Yaskawa INFORM job: A_ROOF_SIDE_0617_2_PAINT_54.JBI

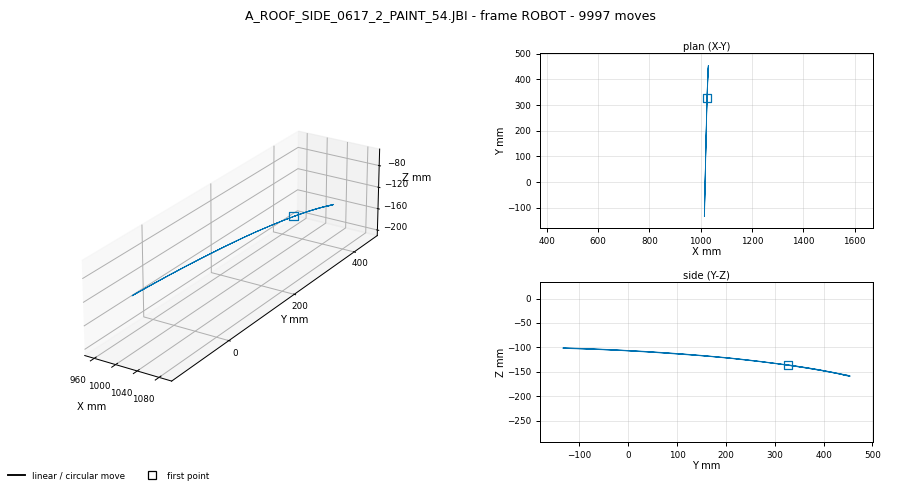
[picture p0: tool path of A_ROOF_SIDE_0617_2_PAINT_54.JBI in frame ROBOT, 9997 of 9997 moves have a stored position in this frame; points joined in program order, loops and branches not executed]
/JOB
//NAME A_ROOF_SIDE_0617_2_PAINT54
//POS
///NPOS 9997,0,0,0,0,0
///TOOL 1
///USER 0
///POSTYPE ROBOT
///RECTAN
///RCONF 1,0,0,0,0,0,0,0,0,0,0,0,0,0,0,0,0,0,0,0,0,0,0,0
C00000=1025.323,327.498,-135.693,171.201,47.894,159.349
C00001=1025.330,327.745,-135.728,171.208,47.893,159.349
C00002=1025.337,327.993,-135.764,171.213,47.892,159.350
C00003=1025.345,328.240,-135.798,171.218,47.891,159.350
C00004=1025.352,328.488,-135.834,171.225,47.891,159.351
C00005=1025.359,328.735,-135.869,171.230,47.890,159.352
C00006=1025.365,328.982,-135.905,171.237,47.889,159.352
C00007=1025.373,329.230,-135.940,171.242,47.888,159.353
C00008=1025.380,329.477,-135.975,171.248,47.888,159.354
C00009=1025.388,329.725,-136.010,171.254,47.886,159.354
C00010=1025.395,329.972,-136.046,171.260,47.886,159.355
C00011=1025.402,330.219,-136.081,171.265,47.885,159.355
C00012=1025.409,330.467,-136.117,171.272,47.885,159.356
C00013=1025.417,330.714,-136.152,171.277,47.884,159.357
C00014=1025.424,330.961,-136.187,171.284,47.883,159.358
C00015=1025.431,331.209,-136.222,171.289,47.883,159.358
C00016=1025.438,331.456,-136.258,171.295,47.882,159.359
C00017=1025.445,331.704,-136.294,171.301,47.881,159.359
C00018=1025.453,331.951,-136.328,171.307,47.880,159.360
C00019=1025.461,332.199,-136.365,171.313,47.880,159.361
C00020=1025.467,332.446,-136.400,171.319,47.880,159.361
C00021=1025.475,332.693,-136.436,171.325,47.878,159.362
C00022=1025.482,332.941,-136.471,171.331,47.878,159.363
C00023=1025.489,333.188,-136.507,171.337,47.877,159.363
C00024=1025.497,333.435,-136.542,171.343,47.877,159.364
C00025=1025.505,333.683,-136.578,171.348,47.876,159.365
C00026=1025.512,333.929,-136.614,171.355,47.876,159.365
C00027=1025.519,334.177,-136.649,171.361,47.875,159.366
C00028=1025.526,334.424,-136.685,171.368,47.875,159.367
C00029=1025.534,334.672,-136.721,171.373,47.874,159.368
C00030=1025.540,334.920,-136.758,171.380,47.873,159.368
C00031=1025.547,335.167,-136.793,171.385,47.873,159.369
C00032=1025.555,335.414,-136.830,171.392,47.873,159.370
C00033=1025.562,335.661,-136.865,171.398,47.872,159.371
C00034=1025.574,336.048,-136.922,171.407,47.871,159.372
C00035=1025.586,336.435,-136.978,171.416,47.871,159.373
C00036=1025.597,336.822,-137.034,171.426,47.870,159.374
C00037=1025.608,337.209,-137.091,171.435,47.869,159.375
C00038=1025.616,337.456,-137.127,171.442,47.869,159.376
C00039=1025.623,337.704,-137.163,171.448,47.869,159.376
C00040=1025.631,337.951,-137.199,171.455,47.868,159.377
C00041=1025.638,338.198,-137.235,171.460,47.868,159.378
C00042=1025.646,338.446,-137.272,171.467,47.867,159.379
C00043=1025.654,338.693,-137.308,171.474,47.867,159.380
C00044=1025.661,338.940,-137.344,171.479,47.866,159.380
C00045=1025.668,339.187,-137.380,171.486,47.866,159.381
C00046=1025.676,339.435,-137.416,171.492,47.866,159.382
C00047=1025.684,339.682,-137.452,171.498,47.865,159.383
C00048=1025.691,339.930,-137.489,171.504,47.865,159.383
C00049=1025.698,340.176,-137.526,171.511,47.865,159.384
C00050=1025.706,340.423,-137.562,171.517,47.865,159.385
C00051=1025.713,340.671,-137.598,171.523,47.864,159.386
C00052=1025.721,340.918,-137.636,171.530,47.864,159.387
C00053=1025.728,341.165,-137.672,171.536,47.864,159.387
C00054=1025.735,341.412,-137.708,171.543,47.864,159.388
C00055=1025.743,341.659,-137.745,171.548,47.863,159.389
C00056=1025.750,341.907,-137.782,171.555,47.863,159.390
C00057=1025.758,342.154,-137.818,171.561,47.863,159.391
C00058=1025.765,342.401,-137.855,171.568,47.863,159.392
C00059=1025.773,342.649,-137.891,171.575,47.862,159.392
C00060=1025.781,342.896,-137.928,171.581,47.863,159.393
C00061=1025.788,343.143,-137.965,171.587,47.862,159.394
C00062=1025.796,343.390,-138.002,171.593,47.862,159.395
C00063=1025.803,343.638,-138.038,171.600,47.862,159.396
C00064=1025.811,343.885,-138.076,171.607,47.861,159.397
C00065=1025.818,344.131,-138.112,171.613,47.862,159.397
C00066=1025.825,344.379,-138.149,171.619,47.861,159.398
C00067=1025.833,344.625,-138.186,171.626,47.861,159.399
C00068=1025.841,344.872,-138.223,171.632,47.861,159.400
C00069=1025.848,345.120,-138.260,171.639,47.861,159.401
C00070=1025.856,345.367,-138.297,171.645,47.861,159.402
C00071=1025.864,345.615,-138.335,171.652,47.861,159.403
C00072=1025.871,345.862,-138.371,171.658,47.860,159.403
C00073=1025.879,346.109,-138.409,171.664,47.861,159.404
C00074=1025.887,346.356,-138.445,171.671,47.861,159.405
C00075=1025.895,346.603,-138.482,171.678,47.860,159.406
C00076=1025.902,346.850,-138.520,171.685,47.860,159.407
C00077=1025.910,347.097,-138.557,171.691,47.861,159.408
C00078=1025.917,347.345,-138.594,171.698,47.860,159.409
C00079=1025.925,347.591,-138.631,171.705,47.860,159.410
C00080=1025.932,347.839,-138.668,171.711,47.861,159.411
C00081=1025.941,348.086,-138.705,171.718,47.861,159.412
C00082=1025.948,348.333,-138.743,171.725,47.860,159.412
C00083=1025.956,348.580,-138.780,171.732,47.860,159.413
C00084=1025.963,348.827,-138.818,171.738,47.861,159.414
C00085=1025.971,349.074,-138.856,171.745,47.861,159.415
C00086=1025.979,349.321,-138.893,171.752,47.861,159.416
C00087=1025.986,349.568,-138.930,171.758,47.861,159.417
C00088=1025.994,349.816,-138.968,171.765,47.861,159.418
C00089=1026.005,350.185,-139.025,171.775,47.861,159.420
C00090=1026.016,350.531,-139.077,171.784,47.861,159.421
C00091=1026.023,350.754,-139.110,171.790,47.862,159.422
C00092=1026.030,350.977,-139.145,171.796,47.862,159.423
C00093=1026.037,351.199,-139.179,171.802,47.862,159.424
C00094=1026.044,351.423,-139.213,171.809,47.862,159.424
C00095=1026.051,351.645,-139.247,171.815,47.862,159.425
C00096=1026.058,351.868,-139.281,171.821,47.863,159.426
C00097=1026.065,352.090,-139.315,171.827,47.863,159.427
C00098=1026.074,352.338,-139.352,171.834,47.863,159.428
C00099=1026.081,352.584,-139.391,171.841,47.863,159.429
C00100=1026.088,352.831,-139.428,171.848,47.863,159.430
C00101=1026.096,353.079,-139.467,171.855,47.863,159.431
C00102=1026.104,353.325,-139.504,171.861,47.864,159.432
C00103=1026.113,353.573,-139.542,171.869,47.864,159.433
C00104=1026.120,353.820,-139.580,171.876,47.864,159.434
C00105=1026.128,354.066,-139.618,171.883,47.864,159.435
C00106=1026.136,354.314,-139.655,171.890,47.865,159.436
C00107=1026.144,354.560,-139.694,171.897,47.865,159.437
C00108=1026.152,354.808,-139.732,171.904,47.865,159.438
C00109=1026.160,355.054,-139.769,171.910,47.866,159.439
C00110=1026.168,355.302,-139.808,171.917,47.866,159.440
C00111=1026.175,355.548,-139.846,171.924,47.866,159.441
C00112=1026.184,355.795,-139.885,171.932,47.867,159.442
C00113=1026.191,356.042,-139.923,171.939,47.867,159.443
C00114=1026.199,356.289,-139.962,171.946,47.868,159.445
C00115=1026.206,356.536,-139.999,171.953,47.868,159.446
C00116=1026.215,356.783,-140.038,171.960,47.868,159.447
C00117=1026.222,357.030,-140.076,171.967,47.868,159.448
C00118=1026.230,357.277,-140.115,171.975,47.869,159.449
C00119=1026.239,357.524,-140.153,171.981,47.870,159.450
C00120=1026.247,357.771,-140.191,171.988,47.870,159.451
C00121=1026.255,358.018,-140.229,171.995,47.871,159.452
C00122=1026.263,358.265,-140.268,172.002,47.871,159.453
C00123=1026.271,358.511,-140.307,172.010,47.872,159.454
C00124=1026.279,358.758,-140.346,172.017,47.872,159.456
C00125=1026.287,359.005,-140.384,172.024,47.873,159.457
C00126=1026.295,359.252,-140.422,172.031,47.873,159.458
C00127=1026.303,359.499,-140.461,172.039,47.874,159.459
C00128=1026.311,359.746,-140.500,172.046,47.874,159.460
C00129=1026.319,359.992,-140.539,172.053,47.875,159.461
C00130=1026.327,360.239,-140.577,172.060,47.875,159.462
C00131=1026.335,360.487,-140.616,172.068,47.876,159.463
C00132=1026.344,360.733,-140.655,172.075,47.876,159.465
C00133=1026.351,360.980,-140.693,172.083,47.877,159.466
C00134=1026.359,361.227,-140.733,172.090,47.878,159.467
C00135=1026.367,361.474,-140.772,172.097,47.878,159.468
C00136=1026.376,361.720,-140.811,172.105,47.879,159.469
C00137=1026.383,361.967,-140.849,172.112,47.880,159.470
C00138=1026.391,362.214,-140.889,172.119,47.880,159.472
C00139=1026.399,362.461,-140.928,172.127,47.881,159.473
C00140=1026.407,362.708,-140.967,172.134,47.882,159.474
C00141=1026.416,362.954,-141.007,172.143,47.882,159.475
C00142=1026.423,363.202,-141.046,172.150,47.883,159.476
C00143=1026.432,363.448,-141.085,172.157,47.884,159.478
C00144=1026.440,363.694,-141.124,172.165,47.884,159.479
C00145=1026.448,363.941,-141.163,172.172,47.885,159.480
C00146=1026.456,364.188,-141.202,172.180,47.886,159.481
C00147=1026.464,364.435,-141.242,172.187,47.887,159.483
C00148=1026.472,364.682,-141.281,172.194,47.888,159.484
C00149=1026.481,364.928,-141.321,172.202,47.888,159.485
C00150=1026.489,365.155,-141.356,172.209,47.889,159.486
C00151=1026.495,365.381,-141.393,172.216,47.890,159.487
C00152=1026.503,365.606,-141.429,172.223,47.891,159.488
C00153=1026.511,365.833,-141.465,172.230,47.891,159.490
C00154=1026.518,366.059,-141.501,172.237,47.892,159.491
C00155=1026.526,366.284,-141.538,172.244,47.893,159.492
C00156=1026.534,366.511,-141.573,172.251,47.893,159.493
C00157=1026.542,366.737,-141.609,172.259,47.895,159.494
C00158=1026.549,366.984,-141.649,172.266,47.895,159.496
C00159=1026.558,367.230,-141.689,172.274,47.897,159.497
C00160=1026.567,367.477,-141.729,172.281,47.897,159.498
C00161=1026.575,367.723,-141.768,172.290,47.898,159.499
C00162=1026.583,367.970,-141.808,172.297,47.899,159.501
C00163=1026.592,368.218,-141.848,172.305,47.900,159.502
C00164=1026.600,368.464,-141.887,172.312,47.901,159.503
C00165=1026.609,368.710,-141.927,172.321,47.902,159.505
C00166=1026.617,368.957,-141.967,172.328,47.903,159.506
C00167=1026.625,369.204,-142.006,172.336,47.903,159.507
C00168=1026.633,369.450,-142.047,172.344,47.905,159.509
C00169=1026.642,369.698,-142.087,172.352,47.906,159.510
C00170=1026.650,369.943,-142.127,172.360,47.907,159.511
C00171=1026.658,370.190,-142.167,172.368,47.908,159.513
C00172=1026.667,370.436,-142.207,172.375,47.909,159.514
C00173=1026.675,370.684,-142.247,172.384,47.910,159.516
C00174=1026.683,370.930,-142.288,172.392,47.911,159.517
C00175=1026.692,371.176,-142.328,172.399,47.912,159.518
C00176=1026.700,371.423,-142.368,172.408,47.913,159.520
C00177=1026.709,371.670,-142.408,172.415,47.914,159.521
C00178=1026.717,371.916,-142.449,172.423,47.915,159.522
C00179=1026.726,372.163,-142.488,172.432,47.917,159.524
C00180=1026.734,372.410,-142.529,172.440,47.918,159.525
C00181=1026.742,372.656,-142.570,172.447,47.919,159.527
C00182=1026.752,372.903,-142.610,172.456,47.920,159.528
C00183=1026.760,373.149,-142.651,172.464,47.922,159.529
C00184=1026.768,373.395,-142.691,172.472,47.923,159.531
C00185=1026.777,373.643,-142.731,172.480,47.924,159.532
C00186=1026.785,373.889,-142.772,172.488,47.926,159.534
C00187=1026.794,374.135,-142.812,172.497,47.926,159.535
C00188=1026.802,374.382,-142.853,172.504,47.928,159.537
C00189=1026.811,374.628,-142.893,172.513,47.929,159.538
C00190=1026.820,374.875,-142.934,172.521,47.930,159.540
C00191=1026.828,375.122,-142.975,172.530,47.931,159.541
C00192=1026.838,375.368,-143.016,172.537,47.933,159.542
C00193=1026.846,375.614,-143.057,172.546,47.934,159.544
C00194=1026.855,375.861,-143.097,172.554,47.935,159.545
C00195=1026.863,376.107,-143.138,172.563,47.937,159.547
C00196=1026.872,376.354,-143.179,172.571,47.938,159.548
C00197=1026.881,376.601,-143.219,172.580,47.939,159.550
C00198=1026.890,376.846,-143.261,172.588,47.941,159.551
C00199=1026.899,377.093,-143.301,172.597,47.942,159.553
C00200=1026.908,377.340,-143.342,172.604,47.943,159.554
C00201=1026.916,377.586,-143.383,172.613,47.945,159.556
C00202=1026.925,377.833,-143.424,172.622,47.946,159.558
C00203=1026.933,378.079,-143.466,172.630,47.948,159.559
C00204=1026.942,378.325,-143.507,172.639,47.949,159.561
C00205=1026.950,378.572,-143.548,172.647,47.951,159.562
C00206=1026.959,378.818,-143.590,172.656,47.952,159.564
C00207=1026.967,379.064,-143.631,172.664,47.954,159.565
C00208=1026.976,379.311,-143.672,172.673,47.955,159.567
C00209=1026.985,379.557,-143.714,172.682,47.957,159.569
C00210=1026.994,379.794,-143.753,172.690,47.958,159.570
C00211=1027.002,380.030,-143.793,172.698,47.960,159.572
C00212=1027.011,380.266,-143.833,172.706,47.961,159.573
C00213=1027.018,380.504,-143.873,172.714,47.963,159.575
C00214=1027.028,380.741,-143.914,172.723,47.964,159.576
C00215=1027.036,380.978,-143.953,172.731,47.966,159.578
C00216=1027.045,381.214,-143.993,172.739,47.968,159.579
C00217=1027.053,381.450,-144.033,172.748,47.969,159.581
C00218=1027.062,381.696,-144.075,172.757,47.970,159.583
C00219=1027.071,381.943,-144.116,172.766,47.973,159.584
C00220=1027.080,382.189,-144.158,172.775,47.974,159.586
C00221=1027.089,382.436,-144.200,172.784,47.976,159.588
C00222=1027.098,382.682,-144.241,172.793,47.977,159.589
C00223=1027.107,382.928,-144.283,172.801,47.979,159.591
C00224=1027.116,383.175,-144.325,172.810,47.981,159.593
C00225=1027.125,383.421,-144.367,172.819,47.982,159.594
C00226=1027.134,383.667,-144.409,172.828,47.984,159.596
C00227=1027.143,383.913,-144.451,172.837,47.986,159.598
C00228=1027.152,384.159,-144.492,172.845,47.988,159.599
C00229=1027.161,384.407,-144.535,172.854,47.989,159.601
C00230=1027.171,384.652,-144.577,172.864,47.991,159.603
C00231=1027.180,384.899,-144.619,172.873,47.993,159.604
C00232=1027.188,385.145,-144.660,172.882,47.995,159.606
C00233=1027.198,385.391,-144.703,172.891,47.996,159.608
C00234=1027.207,385.637,-144.745,172.900,47.998,159.610
C00235=1027.216,385.884,-144.787,172.909,48.001,159.611
C00236=1027.226,386.130,-144.828,172.918,48.002,159.613
C00237=1027.235,386.375,-144.871,172.927,48.004,159.615
C00238=1027.244,386.622,-144.913,172.936,48.006,159.617
C00239=1027.253,386.869,-144.956,172.946,48.008,159.618
C00240=1027.263,387.114,-144.998,172.955,48.010,159.620
C00241=1027.272,387.360,-145.041,172.964,48.012,159.622
C00242=1027.280,387.607,-145.083,172.974,48.014,159.624
C00243=1027.290,387.853,-145.126,172.983,48.016,159.626
C00244=1027.299,388.099,-145.168,172.992,48.018,159.628
C00245=1027.308,388.345,-145.211,173.001,48.019,159.629
C00246=1027.318,388.591,-145.254,173.011,48.021,159.631
C00247=1027.327,388.837,-145.297,173.020,48.023,159.633
C00248=1027.337,389.084,-145.339,173.030,48.025,159.635
C00249=1027.346,389.329,-145.382,173.039,48.027,159.637
C00250=1027.355,389.575,-145.424,173.049,48.030,159.639
C00251=1027.364,389.822,-145.468,173.058,48.032,159.640
C00252=1027.373,390.068,-145.510,173.067,48.034,159.642
C00253=1027.383,390.314,-145.554,173.077,48.036,159.644
C00254=1027.392,390.559,-145.597,173.086,48.038,159.646
C00255=1027.402,390.806,-145.640,173.097,48.040,159.648
C00256=1027.410,391.052,-145.683,173.106,48.042,159.650
C00257=1027.421,391.298,-145.726,173.115,48.045,159.652
C00258=1027.430,391.543,-145.768,173.125,48.047,159.654
C00259=1027.439,391.790,-145.812,173.135,48.049,159.656
C00260=1027.448,392.035,-145.855,173.144,48.051,159.658
C00261=1027.458,392.282,-145.898,173.155,48.053,159.660
C00262=1027.468,392.528,-145.942,173.164,48.055,159.661
C00263=1027.477,392.774,-145.984,173.174,48.058,159.664
C00264=1027.486,393.020,-146.028,173.183,48.061,159.666
C00265=1027.496,393.266,-146.072,173.193,48.063,159.667
C00266=1027.506,393.512,-146.115,173.203,48.065,159.669
C00267=1027.515,393.758,-146.159,173.213,48.067,159.671
C00268=1027.525,394.004,-146.203,173.222,48.070,159.673
C00269=1027.534,394.250,-146.245,173.232,48.072,159.675
C00270=1027.544,394.513,-146.293,173.243,48.074,159.678
C00271=1027.555,394.776,-146.339,173.254,48.077,159.680
C00272=1027.565,395.040,-146.385,173.265,48.079,159.682
C00273=1027.575,395.303,-146.433,173.275,48.082,159.684
C00274=1027.585,395.549,-146.477,173.285,48.084,159.686
C00275=1027.594,395.795,-146.520,173.295,48.087,159.688
C00276=1027.604,396.041,-146.565,173.305,48.089,159.690
C00277=1027.614,396.287,-146.608,173.315,48.092,159.692
C00278=1027.623,396.533,-146.652,173.326,48.094,159.694
C00279=1027.633,396.779,-146.696,173.336,48.097,159.697
C00280=1027.643,397.025,-146.740,173.346,48.100,159.699
C00281=1027.653,397.270,-146.784,173.356,48.102,159.701
C00282=1027.663,397.516,-146.828,173.366,48.105,159.703
C00283=1027.673,397.762,-146.872,173.377,48.107,159.705
C00284=1027.683,398.007,-146.916,173.387,48.109,159.707
C00285=1027.692,398.253,-146.961,173.398,48.112,159.709
C00286=1027.702,398.499,-147.004,173.407,48.115,159.711
C00287=1027.712,398.745,-147.049,173.418,48.117,159.713
C00288=1027.721,398.991,-147.093,173.428,48.120,159.716
C00289=1027.732,399.236,-147.137,173.439,48.122,159.718
C00290=1027.741,399.482,-147.182,173.449,48.125,159.720
C00291=1027.751,399.728,-147.227,173.460,48.128,159.722
C00292=1027.761,399.974,-147.271,173.471,48.130,159.725
C00293=1027.772,400.219,-147.316,173.481,48.134,159.727
C00294=1027.781,400.465,-147.360,173.491,48.136,159.729
C00295=1027.791,400.711,-147.405,173.501,48.139,159.731
C00296=1027.801,400.957,-147.450,173.513,48.142,159.733
C00297=1027.811,401.203,-147.495,173.523,48.144,159.736
C00298=1027.820,401.448,-147.539,173.533,48.147,159.738
C00299=1027.831,401.693,-147.584,173.544,48.150,159.740
C00300=1027.841,401.939,-147.629,173.555,48.153,159.742
C00301=1027.851,402.185,-147.674,173.566,48.155,159.745
C00302=1027.861,402.431,-147.718,173.577,48.159,159.747
C00303=1027.871,402.677,-147.764,173.588,48.161,159.749
C00304=1027.881,402.922,-147.808,173.599,48.164,159.752
C00305=1027.891,403.168,-147.854,173.609,48.167,159.754
C00306=1027.901,403.413,-147.899,173.620,48.170,159.756
C00307=1027.911,403.659,-147.944,173.631,48.173,159.759
C00308=1027.921,403.905,-147.989,173.642,48.176,159.761
C00309=1027.931,404.150,-148.035,173.653,48.179,159.763
C00310=1027.941,404.396,-148.080,173.664,48.182,159.766
C00311=1027.951,404.641,-148.125,173.674,48.185,159.768
C00312=1027.962,404.887,-148.171,173.686,48.188,159.771
C00313=1027.972,405.133,-148.217,173.697,48.191,159.773
C00314=1027.982,405.378,-148.261,173.708,48.194,159.775
C00315=1027.993,405.624,-148.307,173.719,48.197,159.778
C00316=1028.003,405.870,-148.352,173.730,48.200,159.780
C00317=1028.013,406.115,-148.398,173.742,48.203,159.783
C00318=1028.024,406.361,-148.444,173.753,48.206,159.785
C00319=1028.034,406.606,-148.490,173.764,48.209,159.787
C00320=1028.044,406.852,-148.535,173.776,48.212,159.790
C00321=1028.055,407.097,-148.581,173.787,48.216,159.793
C00322=1028.065,407.343,-148.626,173.798,48.219,159.795
C00323=1028.076,407.589,-148.672,173.810,48.222,159.797
C00324=1028.086,407.834,-148.718,173.821,48.225,159.800
C00325=1028.097,408.080,-148.764,173.833,48.228,159.802
C00326=1028.107,408.325,-148.810,173.844,48.232,159.805
C00327=1028.118,408.570,-148.856,173.855,48.235,159.807
C00328=1028.128,408.816,-148.902,173.867,48.237,159.810
C00329=1028.139,409.061,-148.947,173.879,48.241,159.812
C00330=1028.151,409.347,-149.001,173.892,48.245,159.815
C00331=1028.164,409.633,-149.055,173.906,48.249,159.818
C00332=1028.176,409.918,-149.109,173.919,48.253,159.821
C00333=1028.189,410.203,-149.162,173.933,48.256,159.824
C00334=1028.199,410.448,-149.209,173.945,48.260,159.827
C00335=1028.210,410.693,-149.255,173.956,48.263,159.830
C00336=1028.221,410.939,-149.301,173.969,48.267,159.832
C00337=1028.231,411.184,-149.348,173.980,48.270,159.835
C00338=1028.241,411.430,-149.394,173.992,48.273,159.838
C00339=1028.252,411.675,-149.441,174.005,48.277,159.840
C00340=1028.263,411.921,-149.489,174.016,48.281,159.843
C00341=1028.274,412.166,-149.534,174.028,48.284,159.846
C00342=1028.284,412.412,-149.582,174.041,48.288,159.848
C00343=1028.295,412.657,-149.628,174.052,48.291,159.851
C00344=1028.306,412.902,-149.675,174.065,48.294,159.854
C00345=1028.317,413.148,-149.722,174.077,48.298,159.856
C00346=1028.327,413.393,-149.769,174.089,48.302,159.859
C00347=1028.339,413.638,-149.816,174.101,48.305,159.862
C00348=1028.349,413.884,-149.863,174.114,48.308,159.865
C00349=1028.360,414.129,-149.910,174.125,48.312,159.867
C00350=1028.372,414.374,-149.957,174.138,48.316,159.870
C00351=1028.382,414.620,-150.004,174.150,48.319,159.873
C00352=1028.393,414.865,-150.051,174.163,48.324,159.876
C00353=1028.405,415.110,-150.098,174.175,48.327,159.879
C00354=1028.415,415.356,-150.146,174.188,48.331,159.882
C00355=1028.426,415.601,-150.193,174.200,48.334,159.884
C00356=1028.438,415.846,-150.240,174.212,48.338,159.887
C00357=1028.449,416.092,-150.288,174.225,48.342,159.890
C00358=1028.460,416.337,-150.335,174.238,48.346,159.893
C00359=1028.471,416.582,-150.383,174.251,48.349,159.896
C00360=1028.482,416.826,-150.430,174.263,48.353,159.899
C00361=1028.493,417.072,-150.478,174.276,48.357,159.902
C00362=1028.504,417.318,-150.526,174.289,48.361,159.905
C00363=1028.516,417.563,-150.574,174.302,48.365,159.908
C00364=1028.526,417.807,-150.622,174.314,48.369,159.910
C00365=1028.538,418.053,-150.669,174.327,48.373,159.913
C00366=1028.549,418.298,-150.717,174.340,48.377,159.916
C00367=1028.560,418.544,-150.765,174.353,48.381,159.919
C00368=1028.571,418.788,-150.813,174.366,48.384,159.922
C00369=1028.583,419.033,-150.861,174.379,48.388,159.925
C00370=1028.594,419.279,-150.909,174.392,48.392,159.928
C00371=1028.605,419.524,-150.957,174.406,48.396,159.931
C00372=1028.617,419.769,-151.006,174.419,48.400,159.934
C00373=1028.629,420.014,-151.054,174.432,48.405,159.938
C00374=1028.640,420.259,-151.102,174.445,48.409,159.941
C00375=1028.651,420.504,-151.150,174.459,48.413,159.944
C00376=1028.663,420.749,-151.199,174.472,48.417,159.947
C00377=1028.674,420.994,-151.247,174.485,48.420,159.950
C00378=1028.686,421.239,-151.295,174.498,48.425,159.953
C00379=1028.697,421.484,-151.344,174.512,48.429,159.956
C00380=1028.709,421.729,-151.393,174.526,48.433,159.959
C00381=1028.721,421.974,-151.441,174.539,48.437,159.962
C00382=1028.733,422.219,-151.490,174.553,48.442,159.966
C00383=1028.744,422.465,-151.538,174.566,48.446,159.969
C00384=1028.755,422.709,-151.587,174.580,48.450,159.972
C00385=1028.768,422.954,-151.636,174.594,48.454,159.975
C00386=1028.779,423.199,-151.685,174.607,48.459,159.978
C00387=1028.791,423.444,-151.734,174.622,48.462,159.982
C00388=1028.802,423.689,-151.783,174.635,48.467,159.985
C00389=1028.814,423.934,-151.832,174.649,48.471,159.988
C00390=1028.828,424.230,-151.891,174.666,48.476,159.992
C00391=1028.842,424.525,-151.950,174.683,48.482,159.996
C00392=1028.857,424.821,-152.010,174.699,48.488,160.000
C00393=1028.871,425.117,-152.069,174.717,48.493,160.004
C00394=1028.883,425.361,-152.119,174.730,48.497,160.007
C00395=1028.895,425.606,-152.168,174.745,48.501,160.011
C00396=1028.907,425.851,-152.217,174.759,48.505,160.014
C00397=1028.919,426.096,-152.267,174.773,48.510,160.018
C00398=1028.932,426.341,-152.316,174.788,48.515,160.021
C00399=1028.943,426.585,-152.366,174.802,48.520,160.024
C00400=1028.956,426.830,-152.416,174.817,48.524,160.028
C00401=1028.967,427.076,-152.466,174.831,48.528,160.031
C00402=1028.979,427.320,-152.516,174.846,48.533,160.035
C00403=1028.991,427.565,-152.566,174.860,48.538,160.038
C00404=1029.003,427.810,-152.616,174.875,48.543,160.042
C00405=1029.015,428.054,-152.666,174.890,48.547,160.045
C00406=1029.027,428.298,-152.716,174.905,48.552,160.049
C00407=1029.040,428.543,-152.766,174.919,48.556,160.052
C00408=1029.052,428.788,-152.816,174.933,48.561,160.056
C00409=1029.064,429.033,-152.866,174.948,48.566,160.059
C00410=1029.076,429.278,-152.916,174.963,48.571,160.063
C00411=1029.089,429.522,-152.967,174.978,48.575,160.066
C00412=1029.101,429.766,-153.017,174.993,48.580,160.070
C00413=1029.113,430.011,-153.067,175.008,48.585,160.074
C00414=1029.125,430.255,-153.118,175.023,48.590,160.077
C00415=1029.137,430.500,-153.168,175.038,48.595,160.081
C00416=1029.151,430.745,-153.219,175.053,48.599,160.085
C00417=1029.163,430.990,-153.270,175.070,48.604,160.088
C00418=1029.175,431.234,-153.320,175.085,48.609,160.092
C00419=1029.188,431.479,-153.370,175.100,48.614,160.096
C00420=1029.200,431.723,-153.421,175.115,48.619,160.099
C00421=1029.213,431.967,-153.472,175.130,48.624,160.103
C00422=1029.226,432.212,-153.523,175.146,48.629,160.107
C00423=1029.239,432.457,-153.574,175.162,48.634,160.111
C00424=1029.251,432.701,-153.624,175.177,48.639,160.114
C00425=1029.264,432.946,-153.675,175.193,48.644,160.118
C00426=1029.277,433.190,-153.726,175.209,48.649,160.122
C00427=1029.289,433.435,-153.778,175.225,48.654,160.126
C00428=1029.302,433.679,-153.829,175.240,48.659,160.130
C00429=1029.315,433.923,-153.880,175.257,48.664,160.134
C00430=1029.328,434.168,-153.931,175.272,48.669,160.137
C00431=1029.340,434.412,-153.984,175.289,48.674,160.141
C00432=1029.354,434.657,-154.035,175.304,48.679,160.145
C00433=1029.367,434.901,-154.086,175.321,48.685,160.149
C00434=1029.380,435.146,-154.137,175.336,48.690,160.153
C00435=1029.392,435.389,-154.190,175.352,48.695,160.157
C00436=1029.405,435.634,-154.241,175.369,48.700,160.161
C00437=1029.419,435.879,-154.293,175.385,48.706,160.165
C00438=1029.431,436.123,-154.345,175.401,48.711,160.169
C00439=1029.444,436.367,-154.397,175.418,48.716,160.173
C00440=1029.458,436.611,-154.449,175.435,48.721,160.177
C00441=1029.471,436.856,-154.501,175.451,48.727,160.181
C00442=1029.484,437.099,-154.553,175.468,48.732,160.185
C00443=1029.497,437.344,-154.605,175.484,48.738,160.190
C00444=1029.510,437.588,-154.657,175.501,48.743,160.194
C00445=1029.524,437.832,-154.709,175.517,48.748,160.198
C00446=1029.536,438.077,-154.761,175.534,48.754,160.202
C00447=1029.550,438.321,-154.814,175.552,48.759,160.206
C00448=1029.564,438.565,-154.866,175.569,48.765,160.210
C00449=1029.576,438.810,-154.918,175.586,48.770,160.215
C00450=1029.590,439.053,-154.971,175.603,48.776,160.219
C00451=1029.604,439.296,-155.023,175.620,48.781,160.223
C00452=1029.617,439.539,-155.075,175.637,48.787,160.227
C00453=1029.630,439.783,-155.129,175.654,48.792,160.231
C00454=1029.643,440.026,-155.181,175.672,48.798,160.236
C00455=1029.657,440.270,-155.233,175.689,48.803,160.240
C00456=1029.671,440.512,-155.286,175.706,48.809,160.244
C00457=1029.684,440.756,-155.339,175.724,48.815,160.249
C00458=1029.697,441.000,-155.392,175.741,48.821,160.253
C00459=1029.712,441.244,-155.445,175.759,48.826,160.257
C00460=1029.725,441.488,-155.498,175.777,48.832,160.262
C00461=1029.739,441.732,-155.551,175.795,48.837,160.266
C00462=1029.753,441.976,-155.605,175.812,48.844,160.271
C00463=1029.767,442.219,-155.658,175.831,48.849,160.275
C00464=1029.780,442.464,-155.711,175.848,48.856,160.280
C00465=1029.794,442.707,-155.765,175.866,48.861,160.284
C00466=1029.809,442.950,-155.818,175.884,48.867,160.289
C00467=1029.823,443.193,-155.871,175.903,48.872,160.293
C00468=1029.837,443.436,-155.923,175.920,48.878,160.298
C00469=1029.852,443.681,-155.976,175.939,48.884,160.302
C00470=1029.867,443.923,-156.029,175.957,48.890,160.307
C00471=1029.884,444.167,-156.080,175.976,48.895,160.311
C00472=1029.900,444.410,-156.132,175.994,48.901,160.316
C00473=1029.918,444.655,-156.182,176.013,48.906,160.320
C00474=1029.935,444.898,-156.232,176.032,48.911,160.325
C00475=1029.952,445.142,-156.282,176.050,48.917,160.329
C00476=1029.971,445.386,-156.332,176.069,48.922,160.334
C00477=1029.990,445.630,-156.381,176.088,48.926,160.338
C00478=1030.009,445.873,-156.430,176.108,48.932,160.343
C00479=1030.029,446.118,-156.478,176.127,48.936,160.347
C00480=1030.049,446.362,-156.526,176.146,48.941,160.351
C00481=1030.070,446.607,-156.573,176.165,48.946,160.356
C00482=1030.093,446.877,-156.626,176.186,48.951,160.361
C00483=1030.118,447.148,-156.678,176.208,48.956,160.366
C00484=1030.143,447.418,-156.729,176.230,48.961,160.371
C00485=1030.169,447.689,-156.780,176.251,48.966,160.375
C00486=1030.191,447.933,-156.825,176.271,48.971,160.380
C00487=1030.216,448.178,-156.869,176.291,48.975,160.384
C00488=1030.240,448.423,-156.914,176.311,48.979,160.389
C00489=1030.265,448.668,-156.958,176.331,48.984,160.393
C00490=1030.290,448.913,-157.002,176.351,48.988,160.397
C00491=1030.316,449.158,-157.045,176.372,48.992,160.402
C00492=1030.342,449.403,-157.087,176.392,48.995,160.406
C00493=1030.369,449.648,-157.130,176.413,48.999,160.411
C00494=1030.397,449.893,-157.172,176.433,49.004,160.415
C00495=1030.424,450.139,-157.214,176.453,49.007,160.419
C00496=1030.453,450.384,-157.256,176.474,49.011,160.424
C00497=1030.481,450.629,-157.297,176.495,49.015,160.428
C00498=1030.511,450.875,-157.337,176.515,49.018,160.432
C00499=1030.540,451.120,-157.376,176.536,49.022,160.437
C00500=1030.570,451.366,-157.416,176.557,49.025,160.441
C00501=1030.601,451.611,-157.456,176.579,49.029,160.445
C00502=1030.633,451.857,-157.494,176.599,49.032,160.450
C00503=1030.665,452.103,-157.533,176.621,49.035,160.454
C00504=1030.696,452.348,-157.571,176.643,49.038,160.458
C00505=1030.729,452.593,-157.608,176.664,49.042,160.463
C00506=1030.763,452.839,-157.645,176.685,49.045,160.467
C00507=1030.796,453.086,-157.682,176.706,49.048,160.471
C00508=1030.831,453.331,-157.719,176.728,49.051,160.476
C00509=1030.885,453.721,-157.775,176.763,49.055,160.482
C00510=1030.606,453.791,-158.108,176.767,49.118,160.503
C00511=1030.556,453.443,-158.058,176.736,49.114,160.497
C00512=1030.523,453.198,-158.022,176.713,49.112,160.492
C00513=1030.488,452.952,-157.985,176.692,49.109,160.488
C00514=1030.455,452.706,-157.948,176.670,49.106,160.484
C00515=1030.422,452.461,-157.911,176.648,49.103,160.479
C00516=1030.389,452.215,-157.873,176.627,49.100,160.475
C00517=1030.357,451.970,-157.835,176.606,49.096,160.471
C00518=1030.326,451.724,-157.797,176.584,49.093,160.467
C00519=1030.295,451.478,-157.758,176.564,49.090,160.462
C00520=1030.264,451.233,-157.718,176.542,49.087,160.458
C00521=1030.234,450.987,-157.679,176.522,49.083,160.454
C00522=1030.205,450.742,-157.639,176.501,49.080,160.449
C00523=1030.176,450.497,-157.598,176.480,49.076,160.445
C00524=1030.148,450.251,-157.557,176.459,49.072,160.440
C00525=1030.119,450.006,-157.515,176.439,49.069,160.436
C00526=1030.092,449.760,-157.474,176.418,49.065,160.432
C00527=1030.065,449.515,-157.431,176.397,49.061,160.427
C00528=1030.038,449.270,-157.388,176.377,49.058,160.423
C00529=1030.012,449.025,-157.346,176.356,49.054,160.419
C00530=1029.986,448.780,-157.302,176.336,49.049,160.414
C00531=1029.962,448.535,-157.258,176.317,49.046,160.410
C00532=1029.936,448.290,-157.214,176.296,49.042,160.406
C00533=1029.912,448.045,-157.169,176.276,49.037,160.401
C00534=1029.888,447.801,-157.124,176.256,49.033,160.397
C00535=1029.866,447.556,-157.079,176.237,49.029,160.392
C00536=1029.842,447.311,-157.033,176.217,49.024,160.388
C00537=1029.821,447.067,-156.986,176.197,49.020,160.383
C00538=1029.798,446.822,-156.939,176.178,49.015,160.379
C00539=1029.777,446.577,-156.893,176.158,49.011,160.375
C00540=1029.756,446.333,-156.845,176.139,49.006,160.370
C00541=1029.736,446.089,-156.797,176.120,49.001,160.366
C00542=1029.717,445.845,-156.749,176.101,48.997,160.361
C00543=1029.697,445.601,-156.700,176.081,48.992,160.357
C00544=1029.678,445.357,-156.651,176.062,48.986,160.352
C00545=1029.659,445.113,-156.601,176.043,48.982,160.348
C00546=1029.641,444.869,-156.552,176.025,48.977,160.344
C00547=1029.624,444.625,-156.502,176.006,48.971,160.339
C00548=1029.607,444.382,-156.450,175.988,48.966,160.335
C00549=1029.590,444.138,-156.399,175.968,48.961,160.330
C00550=1029.575,443.894,-156.347,175.950,48.956,160.326
C00551=1029.559,443.651,-156.296,175.932,48.950,160.321
C00552=1029.544,443.407,-156.244,175.913,48.944,160.317
C00553=1029.529,443.165,-156.191,175.895,48.939,160.312
C00554=1029.515,442.922,-156.138,175.877,48.933,160.308
C00555=1029.501,442.679,-156.084,175.858,48.927,160.303
C00556=1029.487,442.434,-156.031,175.841,48.921,160.299
C00557=1029.473,442.190,-155.978,175.823,48.916,160.294
C00558=1029.459,441.946,-155.924,175.804,48.910,160.290
C00559=1029.446,441.703,-155.871,175.787,48.905,160.285
C00560=1029.432,441.458,-155.818,175.769,48.899,160.281
C00561=1029.418,441.214,-155.765,175.751,48.893,160.276
C00562=1029.405,440.970,-155.712,175.733,48.887,160.272
C00563=1029.391,440.722,-155.658,175.715,48.882,160.268
C00564=1029.377,440.473,-155.604,175.697,48.876,160.263
C00565=1029.363,440.225,-155.550,175.680,48.871,160.259
C00566=1029.349,439.976,-155.496,175.662,48.865,160.254
C00567=1029.334,439.712,-155.439,175.643,48.859,160.250
C00568=1029.320,439.448,-155.382,175.625,48.853,160.245
C00569=1029.305,439.182,-155.324,175.606,48.847,160.241
C00570=1029.290,438.917,-155.267,175.587,48.841,160.236
C00571=1029.277,438.673,-155.215,175.570,48.836,160.232
C00572=1029.264,438.429,-155.162,175.553,48.831,160.228
C00573=1029.250,438.185,-155.110,175.536,48.825,160.223
C00574=1029.237,437.940,-155.058,175.519,48.820,160.219
C00575=1029.224,437.696,-155.005,175.502,48.814,160.215
C00576=1029.210,437.452,-154.953,175.486,48.809,160.211
C00577=1029.198,437.208,-154.901,175.469,48.804,160.207
C00578=1029.184,436.964,-154.849,175.452,48.798,160.203
C00579=1029.171,436.720,-154.797,175.436,48.793,160.199
C00580=1029.158,436.475,-154.745,175.419,48.788,160.195
C00581=1029.144,436.231,-154.693,175.402,48.783,160.191
C00582=1029.132,435.987,-154.641,175.386,48.778,160.186
C00583=1029.119,435.743,-154.589,175.369,48.772,160.182
C00584=1029.106,435.498,-154.538,175.353,48.767,160.178
C00585=1029.093,435.254,-154.486,175.337,48.762,160.175
C00586=1029.080,435.009,-154.434,175.320,48.757,160.171
C00587=1029.067,434.765,-154.383,175.305,48.751,160.167
C00588=1029.054,434.520,-154.332,175.288,48.747,160.163
C00589=1029.041,434.277,-154.280,175.272,48.742,160.159
C00590=1029.029,434.032,-154.228,175.256,48.736,160.155
C00591=1029.016,433.787,-154.178,175.240,48.732,160.151
C00592=1029.002,433.543,-154.126,175.225,48.727,160.147
C00593=1028.990,433.299,-154.075,175.208,48.722,160.143
C00594=1028.977,433.054,-154.024,175.193,48.716,160.139
C00595=1028.964,432.810,-153.973,175.177,48.711,160.136
C00596=1028.952,432.565,-153.921,175.162,48.707,160.132
C00597=1028.939,432.320,-153.870,175.145,48.702,160.128
C00598=1028.927,432.076,-153.820,175.130,48.697,160.124
C00599=1028.914,431.831,-153.769,175.115,48.692,160.121
C00600=1028.901,431.587,-153.719,175.098,48.687,160.117
C00601=1028.888,431.342,-153.667,175.083,48.683,160.113
C00602=1028.876,431.097,-153.617,175.068,48.678,160.109
C00603=1028.863,430.853,-153.567,175.053,48.673,160.106
C00604=1028.851,430.608,-153.516,175.038,48.668,160.102
C00605=1028.838,430.364,-153.466,175.022,48.664,160.099
C00606=1028.826,430.119,-153.416,175.007,48.659,160.095
C00607=1028.813,429.875,-153.365,174.992,48.654,160.091
C00608=1028.801,429.630,-153.315,174.977,48.649,160.088
C00609=1028.789,429.386,-153.265,174.962,48.645,160.084
C00610=1028.776,429.141,-153.214,174.947,48.640,160.081
C00611=1028.764,428.897,-153.164,174.932,48.636,160.077
C00612=1028.751,428.652,-153.114,174.917,48.631,160.073
C00613=1028.740,428.407,-153.063,174.902,48.626,160.070
C00614=1028.728,428.162,-153.013,174.887,48.622,160.066
C00615=1028.716,427.918,-152.963,174.873,48.617,160.063
C00616=1028.704,427.673,-152.913,174.859,48.612,160.059
C00617=1028.692,427.429,-152.863,174.844,48.608,160.056
C00618=1028.679,427.184,-152.813,174.829,48.603,160.052
C00619=1028.667,426.938,-152.764,174.814,48.599,160.049
C00620=1028.656,426.694,-152.714,174.801,48.594,160.046
C00621=1028.643,426.449,-152.664,174.786,48.590,160.042
C00622=1028.631,426.204,-152.614,174.771,48.586,160.039
C00623=1028.620,425.960,-152.565,174.756,48.581,160.035
C00624=1028.608,425.714,-152.515,174.743,48.577,160.032
C00625=1028.596,425.470,-152.467,174.728,48.572,160.029
C00626=1028.583,425.225,-152.417,174.715,48.568,160.025
C00627=1028.569,424.927,-152.357,174.697,48.563,160.021
C00628=1028.554,424.630,-152.297,174.680,48.558,160.017
C00629=1028.540,424.331,-152.237,174.663,48.552,160.013
C00630=1028.525,424.033,-152.177,174.645,48.547,160.009
C00631=1028.514,423.788,-152.128,174.632,48.543,160.006
C00632=1028.503,423.544,-152.079,174.618,48.539,160.003
C00633=1028.491,423.299,-152.030,174.604,48.534,159.999
C00634=1028.479,423.053,-151.981,174.591,48.530,159.996
C00635=1028.468,422.809,-151.932,174.576,48.526,159.993
C00636=1028.456,422.564,-151.884,174.563,48.522,159.990
C00637=1028.444,422.319,-151.835,174.549,48.517,159.987
C00638=1028.432,422.073,-151.786,174.535,48.514,159.983
C00639=1028.420,421.829,-151.738,174.522,48.509,159.980
C00640=1028.409,421.584,-151.689,174.508,48.505,159.977
C00641=1028.398,421.339,-151.640,174.495,48.501,159.974
C00642=1028.386,421.094,-151.593,174.481,48.497,159.971
C00643=1028.375,420.849,-151.544,174.467,48.493,159.968
C00644=1028.362,420.603,-151.495,174.454,48.489,159.965
C00645=1028.351,420.358,-151.447,174.441,48.485,159.962
C00646=1028.340,420.113,-151.398,174.428,48.481,159.959
C00647=1028.328,419.868,-151.350,174.415,48.477,159.956
C00648=1028.317,419.623,-151.302,174.402,48.474,159.953
C00649=1028.305,419.378,-151.255,174.388,48.470,159.949
C00650=1028.294,419.133,-151.206,174.375,48.466,159.946
C00651=1028.283,418.888,-151.158,174.362,48.462,159.943
C00652=1028.271,418.643,-151.110,174.349,48.458,159.940
C00653=1028.260,418.397,-151.062,174.336,48.454,159.938
C00654=1028.249,418.152,-151.014,174.323,48.450,159.934
C00655=1028.238,417.908,-150.967,174.310,48.446,159.931
C00656=1028.227,417.662,-150.918,174.297,48.443,159.929
C00657=1028.215,417.417,-150.871,174.284,48.439,159.926
C00658=1028.204,417.171,-150.823,174.271,48.435,159.923
C00659=1028.194,416.927,-150.775,174.258,48.431,159.920
C00660=1028.182,416.681,-150.727,174.246,48.428,159.917
C00661=1028.171,416.435,-150.680,174.233,48.424,159.914
C00662=1028.160,416.191,-150.632,174.220,48.420,159.911
C00663=1028.149,415.945,-150.585,174.207,48.417,159.908
C00664=1028.138,415.701,-150.537,174.195,48.412,159.905
C00665=1028.126,415.455,-150.491,174.182,48.409,159.902
C00666=1028.116,415.209,-150.443,174.169,48.405,159.900
C00667=1028.104,414.965,-150.396,174.158,48.402,159.897
C00668=1028.093,414.719,-150.349,174.145,48.398,159.894
C00669=1028.083,414.474,-150.301,174.132,48.395,159.891
C00670=1028.072,414.229,-150.255,174.120,48.391,159.888
C00671=1028.060,413.983,-150.208,174.108,48.388,159.886
C00672=1028.050,413.738,-150.161,174.095,48.384,159.883
C00673=1028.038,413.492,-150.114,174.083,48.381,159.880
C00674=1028.028,413.247,-150.067,174.070,48.377,159.877
C00675=1028.017,413.002,-150.020,174.059,48.373,159.875
C00676=1028.006,412.756,-149.973,174.046,48.370,159.872
C00677=1027.995,412.511,-149.926,174.034,48.367,159.869
C00678=1027.985,412.266,-149.879,174.022,48.364,159.867
C00679=1027.974,412.020,-149.833,174.010,48.360,159.864
C00680=1027.963,411.775,-149.786,173.999,48.357,159.861
C00681=1027.952,411.529,-149.739,173.986,48.353,159.859
C00682=1027.941,411.285,-149.692,173.974,48.350,159.856
C00683=1027.931,411.039,-149.646,173.962,48.346,159.853
C00684=1027.921,410.794,-149.599,173.950,48.343,159.851
C00685=1027.910,410.548,-149.553,173.939,48.340,159.848
C00686=1027.899,410.303,-149.507,173.927,48.336,159.846
C00687=1027.887,410.015,-149.452,173.913,48.333,159.842
C00688=1027.874,409.728,-149.398,173.899,48.329,159.839
C00689=1027.862,409.440,-149.344,173.885,48.325,159.836
C00690=1027.849,409.153,-149.290,173.872,48.321,159.833
C00691=1027.839,408.907,-149.244,173.861,48.318,159.831
C00692=1027.828,408.661,-149.199,173.848,48.315,159.828
C00693=1027.817,408.416,-149.153,173.837,48.312,159.826
C00694=1027.807,408.170,-149.107,173.825,48.309,159.823
C00695=1027.796,407.925,-149.061,173.814,48.305,159.821
C00696=1027.785,407.679,-149.015,173.803,48.303,159.818
C00697=1027.775,407.433,-148.969,173.790,48.300,159.816
C00698=1027.764,407.188,-148.923,173.779,48.296,159.813
C00699=1027.754,406.943,-148.878,173.768,48.294,159.811
C00700=1027.744,406.697,-148.832,173.756,48.290,159.808
C00701=1027.733,406.451,-148.787,173.745,48.287,159.806
C00702=1027.723,406.205,-148.741,173.734,48.284,159.803
C00703=1027.713,405.961,-148.695,173.723,48.281,159.801
C00704=1027.702,405.714,-148.650,173.711,48.278,159.799
C00705=1027.692,405.469,-148.604,173.700,48.275,159.796
C00706=1027.682,405.224,-148.558,173.689,48.272,159.794
C00707=1027.671,404.978,-148.513,173.678,48.269,159.791
C00708=1027.661,404.733,-148.468,173.667,48.267,159.789
C00709=1027.651,404.487,-148.423,173.656,48.264,159.787
C00710=1027.641,404.241,-148.378,173.644,48.261,159.784
C00711=1027.631,403.995,-148.332,173.634,48.257,159.782
C00712=1027.621,403.750,-148.287,173.623,48.255,159.780
C00713=1027.610,403.504,-148.241,173.612,48.252,159.777
C00714=1027.601,403.259,-148.196,173.601,48.249,159.775
C00715=1027.590,403.013,-148.151,173.590,48.246,159.773
C00716=1027.581,402.767,-148.106,173.579,48.244,159.770
C00717=1027.570,402.521,-148.061,173.569,48.241,159.768
C00718=1027.560,402.276,-148.015,173.558,48.238,159.766
C00719=1027.550,402.031,-147.971,173.547,48.235,159.763
C00720=1027.541,401.785,-147.926,173.535,48.232,159.761
C00721=1027.530,401.539,-147.881,173.526,48.230,159.759
C00722=1027.521,401.293,-147.836,173.515,48.227,159.757
C00723=1027.511,401.047,-147.792,173.504,48.224,159.754
C00724=1027.500,400.801,-147.747,173.493,48.222,159.752
C00725=1027.491,400.556,-147.702,173.483,48.219,159.750
C00726=1027.481,400.310,-147.657,173.472,48.216,159.748
C00727=1027.471,400.065,-147.613,173.461,48.214,159.745
C00728=1027.462,399.819,-147.569,173.451,48.211,159.743
C00729=1027.451,399.573,-147.524,173.440,48.208,159.741
C00730=1027.441,399.327,-147.479,173.430,48.205,159.739
C00731=1027.432,399.081,-147.435,173.419,48.203,159.737
C00732=1027.421,398.836,-147.391,173.409,48.201,159.735
C00733=1027.412,398.590,-147.347,173.399,48.198,159.732
C00734=1027.402,398.344,-147.302,173.388,48.196,159.730
C00735=1027.392,398.098,-147.258,173.378,48.193,159.728
C00736=1027.382,397.852,-147.214,173.367,48.191,159.726
C00737=1027.373,397.607,-147.169,173.358,48.188,159.724
C00738=1027.363,397.361,-147.126,173.347,48.185,159.722
C00739=1027.353,397.115,-147.082,173.337,48.183,159.720
C00740=1027.343,396.869,-147.038,173.326,48.181,159.717
C00741=1027.333,396.623,-146.993,173.316,48.178,159.715
C00742=1027.323,396.378,-146.950,173.306,48.176,159.713
C00743=1027.314,396.131,-146.906,173.296,48.173,159.711
C00744=1027.304,395.885,-146.862,173.285,48.171,159.709
C00745=1027.294,395.639,-146.818,173.276,48.169,159.707
C00746=1027.285,395.393,-146.774,173.265,48.167,159.705
C00747=1027.275,395.128,-146.727,173.254,48.164,159.703
C00748=1027.264,394.863,-146.680,173.244,48.161,159.701
C00749=1027.254,394.597,-146.633,173.233,48.159,159.698
C00750=1027.243,394.331,-146.586,173.222,48.156,159.696
C00751=1027.233,394.085,-146.542,173.212,48.154,159.694
C00752=1027.224,393.840,-146.498,173.202,48.152,159.692
C00753=1027.215,393.593,-146.456,173.193,48.149,159.690
C00754=1027.205,393.347,-146.411,173.182,48.148,159.688
C00755=1027.196,393.102,-146.368,173.173,48.145,159.686
C00756=1027.187,392.855,-146.325,173.163,48.143,159.684
C00757=1027.176,392.609,-146.281,173.153,48.141,159.682
C00758=1027.167,392.364,-146.239,173.143,48.139,159.680
C00759=1027.158,392.118,-146.195,173.133,48.136,159.678
C00760=1027.148,391.871,-146.152,173.124,48.134,159.677
C00761=1027.139,391.626,-146.108,173.115,48.132,159.675
C00762=1027.129,391.379,-146.065,173.104,48.130,159.673
C00763=1027.120,391.134,-146.023,173.095,48.128,159.671
C00764=1027.111,390.887,-145.979,173.085,48.126,159.669
C00765=1027.101,390.642,-145.937,173.076,48.124,159.667
C00766=1027.092,390.395,-145.894,173.066,48.122,159.665
C00767=1027.083,390.149,-145.851,173.057,48.119,159.663
C00768=1027.073,389.903,-145.807,173.046,48.118,159.661
C00769=1027.064,389.658,-145.765,173.037,48.116,159.659
C00770=1027.055,389.411,-145.721,173.028,48.114,159.658
C00771=1027.045,389.165,-145.679,173.018,48.112,159.656
C00772=1027.036,388.919,-145.636,173.009,48.110,159.654
C00773=1027.026,388.673,-145.594,172.999,48.108,159.652
C00774=1027.018,388.427,-145.551,172.990,48.106,159.650
C00775=1027.008,388.180,-145.508,172.981,48.104,159.648
C00776=1026.999,387.934,-145.466,172.972,48.102,159.647
C00777=1026.990,387.688,-145.424,172.962,48.100,159.645
C00778=1026.981,387.442,-145.381,172.953,48.098,159.643
C00779=1026.971,387.196,-145.338,172.944,48.097,159.641
C00780=1026.962,386.950,-145.295,172.934,48.095,159.639
C00781=1026.953,386.704,-145.254,172.925,48.093,159.638
C00782=1026.944,386.458,-145.211,172.916,48.091,159.636
C00783=1026.934,386.212,-145.168,172.907,48.089,159.634
C00784=1026.925,385.965,-145.127,172.897,48.087,159.632
C00785=1026.916,385.719,-145.084,172.888,48.086,159.631
C00786=1026.906,385.472,-145.042,172.879,48.084,159.629
C00787=1026.897,385.226,-145.001,172.870,48.082,159.627
C00788=1026.888,384.980,-144.958,172.861,48.081,159.625
C00789=1026.879,384.734,-144.916,172.852,48.079,159.624
C00790=1026.870,384.488,-144.875,172.842,48.077,159.622
C00791=1026.861,384.242,-144.832,172.833,48.075,159.620
C00792=1026.852,383.995,-144.791,172.824,48.074,159.619
C00793=1026.843,383.748,-144.748,172.816,48.072,159.617
C00794=1026.834,383.502,-144.707,172.807,48.070,159.615
C00795=1026.824,383.256,-144.664,172.798,48.068,159.613
C00796=1026.816,383.010,-144.623,172.789,48.067,159.612
C00797=1026.807,382.763,-144.581,172.780,48.065,159.610
C00798=1026.798,382.517,-144.539,172.771,48.064,159.609
C00799=1026.789,382.271,-144.497,172.763,48.062,159.607
C00800=1026.780,382.024,-144.456,172.753,48.061,159.605
C00801=1026.771,381.778,-144.414,172.744,48.059,159.604
C00802=1026.763,381.532,-144.373,172.735,48.058,159.602
C00803=1026.753,381.294,-144.333,172.727,48.056,159.600
C00804=1026.745,381.056,-144.292,172.718,48.055,159.599
C00805=1026.736,380.819,-144.253,172.710,48.053,159.597
C00806=1026.727,380.581,-144.212,172.702,48.052,159.596
C00807=1026.719,380.343,-144.172,172.694,48.050,159.594
C00808=1026.710,380.106,-144.132,172.685,48.049,159.593
C00809=1026.702,379.868,-144.092,172.677,48.047,159.591
C00810=1026.693,379.630,-144.052,172.668,48.046,159.590
C00811=1026.685,379.383,-144.011,172.660,48.044,159.588
C00812=1026.676,379.137,-143.970,172.651,48.043,159.586
C00813=1026.667,378.891,-143.928,172.642,48.042,159.585
C00814=1026.659,378.644,-143.887,172.634,48.040,159.583
C00815=1026.650,378.398,-143.845,172.625,48.039,159.582
C00816=1026.641,378.152,-143.804,172.616,48.037,159.580
C00817=1026.633,377.905,-143.763,172.608,48.036,159.579
C00818=1026.624,377.659,-143.721,172.599,48.034,159.577
C00819=1026.616,377.412,-143.681,172.592,48.033,159.576
C00820=1026.607,377.166,-143.639,172.583,48.032,159.574
C00821=1026.599,376.920,-143.598,172.575,48.030,159.572
C00822=1026.589,376.673,-143.558,172.566,48.029,159.571
C00823=1026.581,376.426,-143.517,172.557,48.028,159.569
C00824=1026.572,376.181,-143.476,172.549,48.026,159.568
C00825=1026.563,375.934,-143.435,172.540,48.025,159.566
C00826=1026.555,375.687,-143.394,172.533,48.024,159.565
C00827=1026.546,375.441,-143.354,172.524,48.023,159.563
C00828=1026.537,375.194,-143.313,172.516,48.022,159.562
C00829=1026.528,374.948,-143.273,172.507,48.021,159.561
C00830=1026.520,374.701,-143.232,172.498,48.019,159.559
C00831=1026.511,374.455,-143.192,172.491,48.018,159.558
C00832=1026.502,374.208,-143.151,172.482,48.017,159.556
C00833=1026.494,373.962,-143.110,172.474,48.016,159.555
C00834=1026.485,373.715,-143.070,172.466,48.015,159.553
C00835=1026.477,373.469,-143.029,172.458,48.014,159.552
C00836=1026.468,373.222,-142.989,172.450,48.012,159.551
C00837=1026.460,372.976,-142.948,172.441,48.011,159.549
C00838=1026.451,372.729,-142.907,172.434,48.010,159.548
C00839=1026.442,372.482,-142.868,172.425,48.009,159.546
C00840=1026.434,372.236,-142.827,172.417,48.008,159.545
C00841=1026.425,371.989,-142.787,172.408,48.007,159.543
C00842=1026.417,371.743,-142.746,172.401,48.006,159.542
C00843=1026.409,371.496,-142.707,172.393,48.005,159.541
C00844=1026.400,371.249,-142.666,172.385,48.004,159.539
C00845=1026.392,371.003,-142.625,172.377,48.003,159.538
C00846=1026.383,370.756,-142.586,172.368,48.002,159.536
C00847=1026.375,370.509,-142.545,172.361,48.001,159.535
C00848=1026.366,370.263,-142.506,172.353,47.999,159.534
C00849=1026.358,370.017,-142.465,172.345,47.999,159.532
C00850=1026.351,369.770,-142.425,172.337,47.998,159.531
C00851=1026.342,369.524,-142.385,172.329,47.997,159.530
C00852=1026.334,369.276,-142.345,172.322,47.995,159.528
C00853=1026.325,369.030,-142.305,172.313,47.995,159.527
C00854=1026.317,368.783,-142.265,172.306,47.994,159.526
C00855=1026.309,368.537,-142.226,172.298,47.993,159.524
C00856=1026.300,368.291,-142.185,172.289,47.992,159.523
C00857=1026.292,368.043,-142.145,172.282,47.991,159.522
C00858=1026.283,367.796,-142.106,172.274,47.990,159.521
C00859=1026.275,367.550,-142.067,172.266,47.989,159.519
C00860=1026.266,367.303,-142.027,172.258,47.989,159.518
C00861=1026.258,367.056,-141.987,172.251,47.988,159.517
C00862=1026.250,366.810,-141.948,172.243,47.987,159.515
C00863=1026.242,366.582,-141.911,172.236,47.986,159.514
C00864=1026.234,366.356,-141.875,172.229,47.986,159.513
C00865=1026.227,366.129,-141.839,172.221,47.985,159.512
C00866=1026.219,365.901,-141.802,172.215,47.984,159.511
C00867=1026.211,365.674,-141.767,172.208,47.984,159.510
C00868=1026.204,365.447,-141.730,172.200,47.983,159.508
C00869=1026.197,365.220,-141.693,172.193,47.982,159.507
C00870=1026.188,364.993,-141.657,172.187,47.981,159.506
C00871=1026.180,364.746,-141.617,172.179,47.981,159.505
C00872=1026.172,364.499,-141.579,172.171,47.980,159.504
C00873=1026.164,364.253,-141.540,172.164,47.980,159.502
C00874=1026.156,364.006,-141.500,172.156,47.979,159.501
C00875=1026.148,363.759,-141.460,172.149,47.978,159.500
C00876=1026.140,363.512,-141.422,172.141,47.977,159.499
C00877=1026.132,363.265,-141.382,172.134,47.977,159.498
C00878=1026.123,363.019,-141.343,172.125,47.976,159.496
C00879=1026.115,362.772,-141.304,172.118,47.976,159.495
C00880=1026.107,362.525,-141.265,172.111,47.975,159.494
C00881=1026.099,362.279,-141.226,172.103,47.974,159.493
C00882=1026.091,362.032,-141.187,172.096,47.974,159.492
C00883=1026.083,361.785,-141.148,172.089,47.973,159.490
C00884=1026.075,361.538,-141.108,172.081,47.972,159.489
C00885=1026.067,361.291,-141.069,172.074,47.972,159.488
C00886=1026.059,361.044,-141.031,172.067,47.972,159.487
C00887=1026.051,360.798,-140.992,172.060,47.971,159.486
C00888=1026.043,360.551,-140.953,172.052,47.970,159.485
C00889=1026.035,360.303,-140.914,172.045,47.970,159.483
C00890=1026.028,360.057,-140.875,172.037,47.969,159.482
C00891=1026.019,359.810,-140.836,172.030,47.969,159.481
C00892=1026.011,359.563,-140.798,172.022,47.969,159.480
C00893=1026.003,359.316,-140.759,172.015,47.968,159.479
C00894=1025.994,359.070,-140.721,172.008,47.968,159.478
C00895=1025.986,358.823,-140.682,172.000,47.967,159.477
C00896=1025.978,358.576,-140.643,171.993,47.967,159.476
C00897=1025.971,358.329,-140.605,171.986,47.967,159.475
C00898=1025.962,358.082,-140.567,171.979,47.966,159.473
C00899=1025.955,357.835,-140.528,171.972,47.966,159.472
C00900=1025.947,357.588,-140.490,171.964,47.965,159.471
C00901=1025.939,357.341,-140.451,171.957,47.965,159.470
C00902=1025.931,357.094,-140.413,171.950,47.965,159.469
C00903=1025.923,356.847,-140.374,171.943,47.965,159.468
C00904=1025.915,356.601,-140.336,171.936,47.964,159.467
C00905=1025.907,356.353,-140.297,171.929,47.964,159.466
C00906=1025.899,356.107,-140.260,171.921,47.963,159.465
C00907=1025.891,355.859,-140.222,171.914,47.963,159.464
C00908=1025.884,355.613,-140.184,171.908,47.963,159.463
C00909=1025.875,355.366,-140.145,171.901,47.962,159.462
C00910=1025.868,355.119,-140.107,171.894,47.962,159.461
C00911=1025.860,354.872,-140.068,171.887,47.962,159.460
C00912=1025.852,354.625,-140.031,171.879,47.961,159.458
C00913=1025.844,354.378,-139.993,171.872,47.961,159.457
C00914=1025.836,354.131,-139.954,171.865,47.961,159.457
C00915=1025.828,353.883,-139.916,171.858,47.961,159.456
C00916=1025.821,353.637,-139.878,171.851,47.961,159.455
C00917=1025.812,353.389,-139.841,171.844,47.960,159.453
C00918=1025.804,353.143,-139.803,171.837,47.960,159.452
C00919=1025.797,352.896,-139.765,171.830,47.960,159.451
C00920=1025.788,352.649,-139.727,171.824,47.960,159.450
C00921=1025.781,352.402,-139.690,171.817,47.960,159.449
C00922=1025.773,352.155,-139.651,171.810,47.960,159.448
C00923=1025.766,351.931,-139.617,171.804,47.960,159.448
C00924=1025.759,351.707,-139.583,171.797,47.959,159.447
C00925=1025.752,351.483,-139.549,171.791,47.960,159.446
C00926=1025.745,351.259,-139.515,171.785,47.959,159.445
C00927=1025.738,351.035,-139.481,171.778,47.959,159.444
C00928=1025.730,350.812,-139.447,171.772,47.960,159.443
C00929=1025.724,350.588,-139.412,171.766,47.959,159.442
C00930=1025.717,350.364,-139.378,171.760,47.959,159.441
C00931=1025.709,350.117,-139.341,171.754,47.959,159.441
C00932=1025.701,349.870,-139.304,171.747,47.959,159.440
C00933=1025.694,349.623,-139.266,171.740,47.959,159.439
C00934=1025.686,349.376,-139.228,171.733,47.959,159.438
C00935=1025.678,349.129,-139.191,171.727,47.959,159.437
C00936=1025.671,348.882,-139.153,171.720,47.959,159.436
C00937=1025.664,348.635,-139.116,171.713,47.959,159.435
C00938=1025.656,348.388,-139.079,171.706,47.959,159.434
C00939=1025.648,348.141,-139.041,171.700,47.959,159.433
C00940=1025.641,347.893,-139.003,171.693,47.959,159.432
C00941=1025.633,347.646,-138.966,171.686,47.959,159.431
C00942=1025.625,347.399,-138.929,171.679,47.959,159.430
C00943=1025.617,347.152,-138.892,171.673,47.960,159.429
C00944=1025.609,346.905,-138.855,171.666,47.959,159.429
C00945=1025.602,346.658,-138.818,171.659,47.959,159.428
C00946=1025.594,346.411,-138.781,171.653,47.960,159.427
C00947=1025.587,346.164,-138.744,171.647,47.960,159.426
C00948=1025.579,345.917,-138.707,171.640,47.960,159.425
C00949=1025.571,345.669,-138.669,171.633,47.960,159.424
C00950=1025.564,345.422,-138.633,171.626,47.961,159.423
C00951=1025.556,345.175,-138.596,171.620,47.960,159.422
C00952=1025.548,344.928,-138.558,171.614,47.961,159.422
C00953=1025.541,344.680,-138.522,171.607,47.961,159.421
C00954=1025.534,344.433,-138.484,171.601,47.961,159.420
C00955=1025.526,344.186,-138.448,171.594,47.962,159.419
C00956=1025.518,343.939,-138.411,171.587,47.961,159.418
C00957=1025.511,343.692,-138.374,171.582,47.962,159.417
C00958=1025.504,343.445,-138.338,171.575,47.962,159.417
C00959=1025.496,343.198,-138.301,171.568,47.962,159.416
C00960=1025.489,342.950,-138.264,171.561,47.963,159.415
C00961=1025.481,342.703,-138.227,171.555,47.963,159.414
C00962=1025.474,342.456,-138.190,171.548,47.963,159.413
C00963=1025.466,342.209,-138.154,171.543,47.963,159.412
C00964=1025.458,341.961,-138.117,171.536,47.964,159.412
C00965=1025.451,341.714,-138.080,171.529,47.964,159.411
C00966=1025.443,341.467,-138.044,171.524,47.964,159.410
C00967=1025.436,341.220,-138.008,171.517,47.964,159.409
C00968=1025.428,340.973,-137.971,171.510,47.965,159.408
C00969=1025.421,340.726,-137.934,171.504,47.965,159.407
C00970=1025.413,340.478,-137.898,171.498,47.966,159.407
C00971=1025.406,340.231,-137.862,171.492,47.966,159.406
C00972=1025.399,339.984,-137.824,171.485,47.966,159.405
C00973=1025.391,339.737,-137.788,171.478,47.967,159.404
C00974=1025.384,339.489,-137.752,171.473,47.967,159.404
C00975=1025.376,339.242,-137.716,171.466,47.968,159.403
C00976=1025.368,338.994,-137.680,171.460,47.968,159.402
C00977=1025.361,338.748,-137.644,171.454,47.969,159.401
C00978=1025.354,338.500,-137.607,171.447,47.969,159.400
C00979=1025.346,338.253,-137.571,171.441,47.969,159.400
C00980=1025.339,338.006,-137.535,171.435,47.970,159.399
C00981=1025.331,337.759,-137.499,171.429,47.970,159.398
C00982=1025.324,337.511,-137.463,171.422,47.971,159.397
C00983=1025.317,337.286,-137.430,171.417,47.972,159.397
C00984=1025.310,337.061,-137.396,171.411,47.972,159.396
C00985=1025.304,336.835,-137.364,171.406,47.972,159.395
C00986=1025.297,336.610,-137.331,171.400,47.973,159.395
C00987=1025.290,336.385,-137.298,171.394,47.973,159.394
C00988=1025.284,336.159,-137.265,171.389,47.974,159.394
C00989=1025.277,335.933,-137.233,171.383,47.974,159.393
C00990=1025.270,335.708,-137.200,171.378,47.974,159.392
C00991=1025.263,335.461,-137.164,171.371,47.976,159.392
C00992=1025.255,335.214,-137.128,171.366,47.976,159.391
C00993=1025.248,334.967,-137.092,171.359,47.976,159.390
C00994=1025.241,334.719,-137.056,171.353,47.978,159.389
C00995=1025.234,334.471,-137.020,171.347,47.978,159.389
C00996=1025.227,334.224,-136.984,171.340,47.978,159.388
C00997=1025.219,333.976,-136.949,171.335,47.979,159.387
C00998=1025.212,333.730,-136.913,171.328,47.980,159.387
C00999=1025.205,333.482,-136.876,171.323,47.980,159.386
C01000=1025.198,333.235,-136.841,171.316,47.981,159.385
C01001=1025.189,332.988,-136.806,171.310,47.981,159.384
C01002=1025.183,332.740,-136.771,171.304,47.982,159.384
C01003=1025.175,332.493,-136.734,171.299,47.983,159.383
C01004=1025.168,332.245,-136.699,171.292,47.984,159.383
C01005=1025.161,331.997,-136.664,171.287,47.985,159.382
C01006=1025.153,331.751,-136.628,171.281,47.985,159.381
C01007=1025.146,331.504,-136.593,171.275,47.986,159.381
C01008=1025.139,331.256,-136.557,171.269,47.986,159.380
C01009=1025.132,331.009,-136.522,171.263,47.988,159.379
C01010=1025.124,330.761,-136.487,171.257,47.988,159.379
C01011=1025.117,330.514,-136.451,171.251,47.989,159.378
C01012=1025.109,330.266,-136.416,171.245,47.990,159.377
C01013=1025.102,330.019,-136.381,171.239,47.991,159.377
C01014=1025.096,329.771,-136.345,171.233,47.991,159.376
C01015=1025.088,329.524,-136.309,171.227,47.992,159.375
C01016=1025.081,329.277,-136.275,171.221,47.993,159.375
C01017=1025.074,329.030,-136.240,171.216,47.994,159.374
C01018=1025.066,328.782,-136.204,171.209,47.995,159.374
C01019=1025.060,328.534,-136.169,171.204,47.995,159.373
C01020=1025.053,328.287,-136.133,171.198,47.997,159.372
C01021=1025.045,328.040,-136.099,171.192,47.997,159.372
C01022=1025.038,327.792,-136.063,171.186,47.998,159.371
C01023=1025.031,327.545,-136.028,171.180,47.999,159.371
C01024=1025.024,327.298,-135.993,171.175,48.000,159.370
C01025=1025.016,327.050,-135.958,171.168,48.001,159.369
C01026=1025.009,326.802,-135.923,171.163,48.002,159.369
C01027=1025.002,326.555,-135.888,171.157,48.003,159.368
C01028=1024.995,326.308,-135.854,171.151,48.004,159.368
C01029=1024.987,326.060,-135.819,171.145,48.005,159.367
C01030=1024.980,325.813,-135.784,171.140,48.006,159.367
C01031=1024.972,325.566,-135.750,171.134,48.007,159.366
C01032=1024.965,325.318,-135.715,171.128,48.008,159.365
C01033=1024.958,325.070,-135.680,171.123,48.009,159.365
C01034=1024.950,324.823,-135.646,171.116,48.010,159.364
C01035=1024.943,324.575,-135.611,171.111,48.011,159.364
C01036=1024.936,324.328,-135.577,171.106,48.012,159.363
C01037=1024.929,324.080,-135.542,171.099,48.013,159.363
C01038=1024.921,323.833,-135.507,171.094,48.014,159.362
C01039=1024.914,323.585,-135.473,171.088,48.016,159.362
C01040=1024.907,323.338,-135.438,171.083,48.017,159.361
C01041=1024.900,323.091,-135.403,171.077,48.018,159.361
C01042=1024.893,322.843,-135.370,171.071,48.019,159.360
C01043=1024.886,322.615,-135.338,171.066,48.020,159.360
C01044=1024.880,322.388,-135.306,171.060,48.021,159.359
C01045=1024.873,322.160,-135.274,171.055,48.022,159.359
C01046=1024.867,321.933,-135.242,171.050,48.023,159.358
C01047=1024.859,321.705,-135.212,171.046,48.024,159.358
C01048=1024.853,321.477,-135.179,171.040,48.025,159.357
C01049=1024.847,321.249,-135.148,171.035,48.026,159.357
C01050=1024.840,321.022,-135.116,171.030,48.027,159.356
C01051=1024.833,320.774,-135.082,171.024,48.028,159.356
C01052=1024.826,320.527,-135.047,171.019,48.030,159.355
C01053=1024.819,320.279,-135.013,171.013,48.031,159.355
C01054=1024.811,320.032,-134.978,171.007,48.032,159.354
C01055=1024.805,319.784,-134.944,171.002,48.033,159.354
C01056=1024.797,319.536,-134.910,170.996,48.034,159.353
C01057=1024.791,319.290,-134.876,170.991,48.036,159.353
C01058=1024.784,319.042,-134.842,170.985,48.037,159.352
C01059=1024.777,318.794,-134.808,170.980,48.038,159.352
C01060=1024.769,318.547,-134.773,170.975,48.039,159.351
C01061=1024.763,318.299,-134.739,170.969,48.041,159.351
C01062=1024.756,318.051,-134.705,170.963,48.042,159.351
C01063=1024.748,317.804,-134.671,170.958,48.043,159.350
C01064=1024.741,317.556,-134.637,170.952,48.044,159.350
C01065=1024.735,317.309,-134.602,170.947,48.046,159.349
C01066=1024.727,317.061,-134.568,170.941,48.047,159.349
C01067=1024.721,316.814,-134.535,170.936,48.048,159.348
C01068=1024.714,316.566,-134.501,170.930,48.049,159.348
C01069=1024.707,316.318,-134.467,170.925,48.051,159.347
C01070=1024.700,316.071,-134.433,170.920,48.052,159.347
C01071=1024.693,315.823,-134.398,170.915,48.053,159.346
C01072=1024.686,315.576,-134.364,170.909,48.055,159.346
C01073=1024.679,315.329,-134.330,170.903,48.056,159.345
C01074=1024.673,315.081,-134.296,170.898,48.057,159.345
C01075=1024.666,314.833,-134.262,170.893,48.059,159.345
C01076=1024.659,314.586,-134.229,170.887,48.060,159.344
C01077=1024.652,314.338,-134.195,170.882,48.061,159.344
C01078=1024.645,314.090,-134.161,170.877,48.063,159.343
C01079=1024.638,313.843,-134.127,170.871,48.064,159.343
C01080=1024.632,313.596,-134.093,170.866,48.065,159.342
C01081=1024.625,313.348,-134.059,170.860,48.067,159.342
C01082=1024.618,313.100,-134.025,170.855,48.068,159.342
C01083=1024.611,312.853,-133.992,170.850,48.069,159.341
C01084=1024.605,312.605,-133.958,170.845,48.071,159.341
C01085=1024.598,312.357,-133.924,170.840,48.072,159.340
C01086=1024.591,312.110,-133.891,170.834,48.074,159.340
C01087=1024.584,311.862,-133.857,170.829,48.075,159.340
C01088=1024.578,311.615,-133.823,170.823,48.076,159.339
C01089=1024.571,311.367,-133.789,170.818,48.078,159.339
C01090=1024.564,311.120,-133.755,170.813,48.079,159.338
C01091=1024.558,310.872,-133.722,170.808,48.081,159.338
C01092=1024.551,310.624,-133.688,170.802,48.083,159.338
C01093=1024.545,310.377,-133.654,170.797,48.084,159.337
C01094=1024.537,310.129,-133.622,170.792,48.085,159.337
C01095=1024.530,309.882,-133.588,170.787,48.087,159.336
C01096=1024.523,309.634,-133.555,170.781,48.089,159.336
C01097=1024.515,309.386,-133.522,170.776,48.090,159.336
C01098=1024.509,309.139,-133.489,170.771,48.092,159.335
C01099=1024.502,308.891,-133.456,170.766,48.094,159.335
C01100=1024.494,308.643,-133.423,170.760,48.096,159.335
C01101=1024.488,308.396,-133.390,170.755,48.097,159.334
C01102=1024.481,308.148,-133.356,170.750,48.099,159.334
C01103=1024.474,307.923,-133.327,170.745,48.100,159.334
C01104=1024.468,307.698,-133.297,170.740,48.102,159.333
C01105=1024.462,307.473,-133.267,170.736,48.103,159.333
C01106=1024.456,307.247,-133.237,170.731,48.105,159.333
C01107=1024.449,307.022,-133.207,170.726,48.106,159.332
C01108=1024.443,306.797,-133.177,170.721,48.108,159.332
C01109=1024.436,306.572,-133.147,170.718,48.110,159.332
C01110=1024.430,306.348,-133.118,170.712,48.111,159.332
C01111=1024.423,306.100,-133.084,170.707,48.113,159.331
C01112=1024.417,305.852,-133.052,170.703,48.115,159.331
C01113=1024.409,305.604,-133.019,170.697,48.117,159.331
C01114=1024.403,305.357,-132.986,170.692,48.118,159.330
C01115=1024.396,305.109,-132.953,170.687,48.120,159.330
C01116=1024.389,304.862,-132.921,170.682,48.122,159.330
C01117=1024.382,304.613,-132.887,170.677,48.123,159.329
C01118=1024.375,304.366,-132.855,170.671,48.126,159.329
C01119=1024.368,304.118,-132.822,170.666,48.127,159.329
C01120=1024.362,303.870,-132.789,170.661,48.129,159.329
C01121=1024.355,303.623,-132.757,170.656,48.131,159.328
C01122=1024.348,303.375,-132.724,170.651,48.132,159.328
C01123=1024.341,303.128,-132.691,170.647,48.134,159.328
C01124=1024.334,302.880,-132.659,170.642,48.136,159.327
C01125=1024.327,302.632,-132.625,170.636,48.138,159.327
C01126=1024.321,302.384,-132.593,170.631,48.140,159.327
C01127=1024.313,302.136,-132.560,170.626,48.142,159.327
C01128=1024.307,301.889,-132.527,170.621,48.143,159.326
C01129=1024.301,301.641,-132.495,170.616,48.145,159.326
C01130=1024.294,301.393,-132.463,170.611,48.147,159.326
C01131=1024.287,301.145,-132.430,170.607,48.149,159.325
C01132=1024.280,300.898,-132.398,170.601,48.151,159.325
C01133=1024.274,300.650,-132.365,170.596,48.153,159.325
C01134=1024.267,300.402,-132.332,170.591,48.154,159.325
C01135=1024.260,300.155,-132.300,170.586,48.156,159.324
C01136=1024.254,299.907,-132.267,170.581,48.159,159.324
C01137=1024.247,299.659,-132.235,170.576,48.160,159.324
C01138=1024.240,299.411,-132.203,170.572,48.162,159.324
C01139=1024.234,299.163,-132.170,170.567,48.164,159.323
C01140=1024.227,298.916,-132.138,170.562,48.166,159.323
C01141=1024.220,298.668,-132.105,170.556,48.168,159.323
C01142=1024.214,298.421,-132.072,170.551,48.170,159.322
C01143=1024.207,298.172,-132.041,170.546,48.172,159.322
C01144=1024.201,297.925,-132.008,170.542,48.174,159.322
C01145=1024.194,297.677,-131.975,170.537,48.175,159.322
C01146=1024.188,297.429,-131.944,170.532,48.178,159.322
C01147=1024.181,297.181,-131.911,170.527,48.180,159.321
C01148=1024.174,296.934,-131.879,170.523,48.182,159.321
C01149=1024.168,296.685,-131.846,170.518,48.183,159.321
C01150=1024.161,296.438,-131.814,170.513,48.185,159.321
C01151=1024.154,296.190,-131.781,170.508,48.188,159.320
C01152=1024.148,295.942,-131.749,170.503,48.190,159.320
C01153=1024.142,295.695,-131.717,170.498,48.191,159.320
C01154=1024.135,295.447,-131.685,170.494,48.193,159.320
C01155=1024.129,295.199,-131.653,170.489,48.195,159.320
C01156=1024.122,294.952,-131.620,170.483,48.198,159.319
C01157=1024.116,294.704,-131.588,170.478,48.199,159.319
C01158=1024.110,294.456,-131.556,170.473,48.201,159.319
C01159=1024.103,294.208,-131.524,170.469,48.204,159.319
C01160=1024.097,293.960,-131.491,170.464,48.206,159.318
C01161=1024.089,293.712,-131.460,170.459,48.208,159.318
C01162=1024.083,293.464,-131.428,170.455,48.210,159.318
C01163=1024.078,293.248,-131.400,170.451,48.212,159.318
C01164=1024.072,293.031,-131.372,170.446,48.214,159.318
C01165=1024.065,292.815,-131.344,170.443,48.216,159.318
C01166=1024.060,292.599,-131.317,170.438,48.217,159.317
C01167=1024.054,292.383,-131.289,170.434,48.219,159.317
C01168=1024.048,292.166,-131.261,170.430,48.221,159.317
C01169=1024.043,291.949,-131.233,170.425,48.223,159.317
C01170=1024.037,291.733,-131.206,170.422,48.225,159.317
C01171=1024.030,291.485,-131.174,170.417,48.227,159.317
C01172=1024.023,291.238,-131.142,170.412,48.229,159.316
C01173=1024.017,290.990,-131.110,170.408,48.232,159.316
C01174=1024.010,290.742,-131.079,170.402,48.234,159.316
C01175=1024.004,290.494,-131.047,170.397,48.236,159.316
C01176=1023.997,290.246,-131.016,170.393,48.239,159.316
C01177=1023.990,289.998,-130.984,170.388,48.241,159.316
C01178=1023.983,289.750,-130.953,170.383,48.243,159.315
C01179=1023.977,289.502,-130.922,170.379,48.246,159.315
C01180=1023.971,289.254,-130.890,170.374,48.248,159.315
C01181=1023.964,289.006,-130.858,170.370,48.250,159.315
C01182=1023.957,288.758,-130.827,170.365,48.252,159.315
C01183=1023.951,288.510,-130.795,170.360,48.255,159.315
C01184=1023.944,288.262,-130.764,170.356,48.257,159.315
C01185=1023.937,288.014,-130.732,170.351,48.259,159.315
C01186=1023.930,287.767,-130.701,170.346,48.261,159.314
C01187=1023.924,287.519,-130.670,170.342,48.264,159.314
C01188=1023.918,287.271,-130.638,170.337,48.266,159.314
C01189=1023.911,287.024,-130.607,170.333,48.268,159.314
C01190=1023.904,286.776,-130.576,170.328,48.271,159.314
C01191=1023.898,286.527,-130.544,170.323,48.273,159.314
C01192=1023.892,286.279,-130.513,170.318,48.276,159.314
C01193=1023.885,286.031,-130.481,170.313,48.278,159.314
C01194=1023.878,285.783,-130.450,170.309,48.281,159.313
C01195=1023.872,285.536,-130.419,170.304,48.283,159.313
C01196=1023.865,285.288,-130.388,170.300,48.285,159.313
C01197=1023.859,285.039,-130.357,170.295,48.288,159.313
C01198=1023.852,284.792,-130.326,170.291,48.290,159.313
C01199=1023.845,284.544,-130.295,170.286,48.293,159.313
C01200=1023.838,284.295,-130.264,170.281,48.295,159.313
C01201=1023.832,284.048,-130.233,170.277,48.298,159.313
C01202=1023.826,283.800,-130.201,170.272,48.300,159.313
C01203=1023.819,283.552,-130.171,170.268,48.303,159.313
C01204=1023.812,283.304,-130.140,170.263,48.305,159.312
C01205=1023.805,283.056,-130.109,170.259,48.308,159.312
C01206=1023.799,282.809,-130.078,170.254,48.310,159.312
C01207=1023.793,282.560,-130.047,170.250,48.313,159.312
C01208=1023.786,282.312,-130.016,170.245,48.316,159.312
C01209=1023.779,282.064,-129.986,170.241,48.318,159.312
C01210=1023.772,281.816,-129.954,170.236,48.321,159.312
C01211=1023.766,281.568,-129.924,170.232,48.323,159.312
C01212=1023.760,281.320,-129.892,170.227,48.325,159.312
C01213=1023.753,281.072,-129.862,170.223,48.328,159.312
C01214=1023.747,280.825,-129.831,170.218,48.331,159.312
C01215=1023.740,280.576,-129.801,170.214,48.333,159.312
C01216=1023.733,280.328,-129.769,170.209,48.336,159.312
C01217=1023.727,280.080,-129.738,170.205,48.339,159.312
C01218=1023.721,279.833,-129.707,170.200,48.341,159.312
C01219=1023.714,279.584,-129.677,170.196,48.344,159.312
C01220=1023.708,279.336,-129.646,170.192,48.346,159.312
C01221=1023.701,279.089,-129.615,170.187,48.349,159.311
C01222=1023.694,278.840,-129.585,170.182,48.351,159.311
C01223=1023.690,278.630,-129.559,170.178,48.354,159.311
C01224=1023.684,278.420,-129.532,170.174,48.356,159.311
C01225=1023.679,278.209,-129.507,170.171,48.358,159.311
C01226=1023.673,277.999,-129.481,170.167,48.360,159.311
C01227=1023.667,277.789,-129.455,170.163,48.363,159.311
C01228=1023.662,277.578,-129.429,170.159,48.365,159.311
C01229=1023.657,277.368,-129.403,170.156,48.367,159.311
C01230=1023.651,277.158,-129.376,170.152,48.369,159.311
C01231=1023.645,276.910,-129.346,170.148,48.372,159.311
C01232=1023.638,276.662,-129.316,170.143,48.375,159.311
C01233=1023.632,276.414,-129.285,170.139,48.378,159.311
C01234=1023.625,276.166,-129.255,170.135,48.380,159.311
C01235=1023.618,275.917,-129.225,170.130,48.383,159.311
C01236=1023.612,275.670,-129.194,170.126,48.386,159.311
C01237=1023.605,275.422,-129.163,170.122,48.389,159.311
C01238=1023.599,275.174,-129.134,170.117,48.392,159.311
C01239=1023.592,274.926,-129.103,170.113,48.394,159.311
C01240=1023.586,274.677,-129.072,170.108,48.397,159.311
C01241=1023.579,274.430,-129.042,170.104,48.400,159.311
C01242=1023.573,274.181,-129.012,170.100,48.403,159.311
C01243=1023.566,273.934,-128.982,170.095,48.406,159.311
C01244=1023.560,273.685,-128.951,170.091,48.408,159.311
C01245=1023.553,273.438,-128.921,170.087,48.411,159.311
C01246=1023.547,273.189,-128.891,170.082,48.414,159.311
C01247=1023.540,272.942,-128.861,170.078,48.417,159.311
C01248=1023.534,272.693,-128.830,170.073,48.420,159.311
C01249=1023.528,272.445,-128.801,170.069,48.422,159.311
C01250=1023.521,272.197,-128.770,170.065,48.425,159.311
C01251=1023.515,271.949,-128.741,170.060,48.428,159.311
C01252=1023.508,271.701,-128.710,170.056,48.431,159.311
C01253=1023.502,271.453,-128.680,170.052,48.434,159.311
C01254=1023.495,271.204,-128.650,170.048,48.437,159.311
C01255=1023.489,270.956,-128.620,170.043,48.440,159.311
C01256=1023.483,270.708,-128.590,170.039,48.443,159.311
C01257=1023.476,270.460,-128.560,170.034,48.445,159.311
C01258=1023.470,270.212,-128.529,170.030,48.449,159.311
C01259=1023.463,269.964,-128.500,170.026,48.452,159.311
C01260=1023.457,269.716,-128.471,170.022,48.454,159.311
C01261=1023.450,269.468,-128.440,170.017,48.457,159.311
C01262=1023.444,269.220,-128.410,170.013,48.461,159.311
C01263=1023.437,268.971,-128.381,170.009,48.463,159.311
C01264=1023.431,268.723,-128.350,170.005,48.466,159.311
C01265=1023.425,268.476,-128.321,170.000,48.470,159.312
C01266=1023.418,268.227,-128.291,169.996,48.473,159.312
C01267=1023.412,267.979,-128.261,169.992,48.475,159.312
C01268=1023.405,267.730,-128.231,169.988,48.479,159.312
C01269=1023.399,267.483,-128.202,169.983,48.482,159.312
C01270=1023.393,267.235,-128.171,169.979,48.484,159.312
C01271=1023.386,266.986,-128.142,169.975,48.488,159.312
C01272=1023.379,266.739,-128.112,169.971,48.491,159.312
C01273=1023.373,266.490,-128.083,169.966,48.493,159.312
C01274=1023.367,266.242,-128.052,169.962,48.497,159.312
C01275=1023.360,265.994,-128.023,169.958,48.500,159.312
C01276=1023.353,265.746,-127.993,169.954,48.503,159.312
C01277=1023.347,265.498,-127.964,169.949,48.506,159.312
C01278=1023.341,265.250,-127.935,169.945,48.509,159.313
C01279=1023.334,265.001,-127.904,169.941,48.512,159.312
C01280=1023.328,264.753,-127.875,169.937,48.516,159.313
C01281=1023.322,264.505,-127.846,169.933,48.518,159.313
C01282=1023.315,264.257,-127.817,169.929,48.522,159.313
C01283=1023.304,263.841,-127.767,169.921,48.527,159.313
C01284=1023.294,263.424,-127.717,169.914,48.532,159.313
C01285=1023.283,263.009,-127.668,169.908,48.538,159.313
C01286=1023.272,262.593,-127.619,169.900,48.543,159.313
C01287=1023.266,262.345,-127.589,169.896,48.546,159.313
C01288=1023.259,262.097,-127.560,169.892,48.550,159.314
C01289=1023.252,261.848,-127.531,169.888,48.553,159.314
C01290=1023.247,261.600,-127.501,169.883,48.556,159.314
C01291=1023.240,261.352,-127.472,169.879,48.559,159.314
C01292=1023.234,261.104,-127.443,169.876,48.562,159.314
C01293=1023.227,260.855,-127.413,169.872,48.565,159.314
C01294=1023.221,260.607,-127.384,169.868,48.569,159.314
C01295=1023.215,260.359,-127.355,169.864,48.572,159.315
C01296=1023.209,260.111,-127.326,169.859,48.575,159.315
C01297=1023.202,259.863,-127.298,169.854,48.579,159.315
C01298=1023.195,259.615,-127.269,169.850,48.582,159.315
C01299=1023.188,259.366,-127.239,169.846,48.586,159.315
C01300=1023.182,259.118,-127.210,169.842,48.589,159.315
C01301=1023.175,258.870,-127.182,169.838,48.593,159.315
C01302=1023.169,258.622,-127.153,169.834,48.596,159.316
C01303=1023.162,258.373,-127.123,169.830,48.600,159.316
C01304=1023.155,258.125,-127.095,169.826,48.602,159.316
C01305=1023.149,257.877,-127.066,169.822,48.606,159.316
C01306=1023.143,257.629,-127.037,169.818,48.609,159.316
C01307=1023.136,257.381,-127.008,169.814,48.613,159.316
C01308=1023.129,257.132,-126.980,169.810,48.616,159.316
C01309=1023.123,256.884,-126.950,169.806,48.620,159.317
C01310=1023.117,256.636,-126.921,169.802,48.623,159.317
C01311=1023.110,256.387,-126.892,169.798,48.627,159.317
C01312=1023.103,256.140,-126.864,169.793,48.630,159.317
C01313=1023.097,255.891,-126.836,169.789,48.634,159.317
C01314=1023.091,255.643,-126.807,169.785,48.637,159.317
C01315=1023.084,255.394,-126.778,169.781,48.641,159.318
C01316=1023.077,255.146,-126.749,169.777,48.644,159.318
C01317=1023.071,254.898,-126.720,169.773,48.648,159.318
C01318=1023.065,254.649,-126.691,169.769,48.651,159.318
C01319=1023.058,254.401,-126.663,169.765,48.654,159.318
C01320=1023.052,254.153,-126.634,169.761,48.658,159.318
C01321=1023.046,253.904,-126.606,169.757,48.661,159.319
C01322=1023.039,253.657,-126.577,169.753,48.665,159.319
C01323=1023.033,253.409,-126.548,169.749,48.668,159.319
C01324=1023.026,253.160,-126.519,169.745,48.672,159.319
C01325=1023.020,252.912,-126.491,169.741,48.675,159.319
C01326=1023.014,252.664,-126.462,169.737,48.679,159.320
C01327=1023.008,252.415,-126.434,169.733,48.683,159.320
C01328=1023.001,252.167,-126.405,169.729,48.686,159.320
C01329=1022.994,251.919,-126.376,169.725,48.690,159.320
C01330=1022.988,251.670,-126.348,169.721,48.693,159.320
C01331=1022.982,251.422,-126.319,169.717,48.697,159.321
C01332=1022.975,251.174,-126.291,169.713,48.700,159.321
C01333=1022.969,250.926,-126.262,169.709,48.704,159.321
C01334=1022.963,250.678,-126.233,169.706,48.708,159.321
C01335=1022.956,250.429,-126.206,169.702,48.711,159.321
C01336=1022.950,250.181,-126.177,169.698,48.715,159.322
C01337=1022.944,249.932,-126.148,169.694,48.718,159.322
C01338=1022.938,249.684,-126.119,169.689,48.722,159.322
C01339=1022.927,249.266,-126.072,169.683,48.728,159.322
C01340=1022.917,248.849,-126.023,169.676,48.734,159.323
C01341=1022.905,248.431,-125.976,169.670,48.740,159.323
C01342=1022.895,248.013,-125.927,169.663,48.747,159.323
C01343=1022.888,247.765,-125.900,169.659,48.750,159.324
C01344=1022.883,247.518,-125.871,169.655,48.754,159.324
C01345=1022.877,247.269,-125.843,169.651,48.758,159.324
C01346=1022.870,247.020,-125.815,169.648,48.761,159.324
C01347=1022.864,246.772,-125.786,169.644,48.764,159.325
C01348=1022.858,246.523,-125.758,169.640,48.769,159.325
C01349=1022.851,246.276,-125.729,169.636,48.772,159.325
C01350=1022.845,246.027,-125.701,169.632,48.776,159.325
C01351=1022.840,245.779,-125.673,169.628,48.779,159.325
C01352=1022.833,245.531,-125.644,169.624,48.783,159.326
C01353=1022.827,245.282,-125.616,169.620,48.787,159.326
C01354=1022.821,245.034,-125.588,169.616,48.790,159.326
C01355=1022.814,244.786,-125.559,169.613,48.794,159.326
C01356=1022.808,244.537,-125.531,169.609,48.798,159.327
C01357=1022.803,244.289,-125.503,169.605,48.801,159.327
C01358=1022.796,244.040,-125.475,169.601,48.806,159.327
C01359=1022.790,243.792,-125.446,169.597,48.809,159.327
C01360=1022.784,243.544,-125.418,169.593,48.813,159.328
C01361=1022.777,243.295,-125.390,169.589,48.817,159.328
C01362=1022.771,243.047,-125.363,169.586,48.821,159.328
C01363=1022.765,242.799,-125.335,169.582,48.824,159.328
C01364=1022.758,242.550,-125.307,169.578,48.828,159.329
C01365=1022.752,242.302,-125.278,169.574,48.832,159.329
C01366=1022.745,242.054,-125.250,169.570,48.836,159.329
C01367=1022.739,241.806,-125.223,169.566,48.840,159.329
C01368=1022.733,241.557,-125.194,169.563,48.844,159.330
C01369=1022.727,241.309,-125.167,169.559,48.848,159.330
C01370=1022.721,241.060,-125.138,169.555,48.851,159.330
C01371=1022.715,240.812,-125.111,169.551,48.856,159.331
C01372=1022.708,240.564,-125.083,169.547,48.859,159.331
C01373=1022.702,240.315,-125.055,169.544,48.863,159.331
C01374=1022.695,240.067,-125.027,169.540,48.867,159.331
C01375=1022.690,239.819,-124.999,169.536,48.871,159.332
C01376=1022.683,239.570,-124.971,169.532,48.875,159.332
C01377=1022.677,239.322,-124.944,169.528,48.879,159.332
C01378=1022.670,239.073,-124.916,169.524,48.883,159.333
C01379=1022.664,238.825,-124.889,169.521,48.887,159.333
C01380=1022.658,238.576,-124.861,169.517,48.891,159.333
C01381=1022.652,238.328,-124.833,169.513,48.895,159.333
C01382=1022.645,238.079,-124.806,169.509,48.899,159.334
C01383=1022.639,237.831,-124.778,169.506,48.903,159.334
C01384=1022.632,237.583,-124.750,169.502,48.907,159.335
C01385=1022.626,237.334,-124.723,169.498,48.911,159.335
C01386=1022.620,237.086,-124.696,169.494,48.915,159.335
C01387=1022.614,236.837,-124.668,169.491,48.919,159.335
C01388=1022.607,236.589,-124.640,169.487,48.923,159.336
C01389=1022.601,236.341,-124.613,169.482,48.928,159.336
C01390=1022.595,236.092,-124.586,169.479,48.932,159.336
C01391=1022.588,235.844,-124.558,169.475,48.936,159.337
C01392=1022.582,235.595,-124.531,169.471,48.940,159.337
C01393=1022.575,235.347,-124.504,169.467,48.944,159.337
C01394=1022.569,235.099,-124.476,169.464,48.948,159.338
C01395=1022.564,234.887,-124.453,169.461,48.952,159.338
C01396=1022.558,234.675,-124.429,169.458,48.955,159.338
C01397=1022.553,234.462,-124.405,169.454,48.958,159.338
C01398=1022.547,234.251,-124.383,169.451,48.962,159.339
C01399=1022.542,234.039,-124.359,169.448,48.965,159.339
C01400=1022.536,233.827,-124.336,169.444,48.969,159.339
C01401=1022.532,233.615,-124.313,169.442,48.973,159.340
C01402=1022.526,233.403,-124.289,169.439,48.976,159.340
C01403=1022.520,233.155,-124.262,169.435,48.980,159.340
C01404=1022.514,232.906,-124.234,169.431,48.984,159.341
C01405=1022.507,232.658,-124.207,169.428,48.989,159.341
C01406=1022.501,232.409,-124.180,169.424,48.993,159.341
C01407=1022.494,232.161,-124.152,169.420,48.997,159.342
C01408=1022.489,231.913,-124.126,169.417,49.001,159.342
C01409=1022.482,231.664,-124.098,169.413,49.005,159.342
C01410=1022.476,231.416,-124.071,169.408,49.010,159.343
C01411=1022.470,231.167,-124.044,169.405,49.014,159.343
C01412=1022.463,230.918,-124.017,169.401,49.018,159.343
C01413=1022.457,230.671,-123.989,169.397,49.022,159.344
C01414=1022.451,230.421,-123.962,169.394,49.027,159.344
C01415=1022.445,230.174,-123.935,169.390,49.031,159.345
C01416=1022.438,229.925,-123.908,169.386,49.035,159.345
C01417=1022.432,229.676,-123.881,169.383,49.040,159.345
C01418=1022.426,229.428,-123.853,169.380,49.044,159.346
C01419=1022.420,229.180,-123.827,169.376,49.048,159.346
C01420=1022.413,228.931,-123.799,169.372,49.052,159.346
C01421=1022.408,228.683,-123.772,169.369,49.057,159.347
C01422=1022.400,228.434,-123.746,169.365,49.061,159.347
C01423=1022.394,228.186,-123.719,169.362,49.066,159.348
C01424=1022.388,227.937,-123.692,169.358,49.070,159.348
C01425=1022.382,227.689,-123.665,169.354,49.074,159.348
C01426=1022.376,227.440,-123.637,169.351,49.078,159.349
C01427=1022.370,227.192,-123.611,169.347,49.082,159.349
C01428=1022.363,226.943,-123.584,169.343,49.087,159.350
C01429=1022.357,226.695,-123.557,169.339,49.092,159.350
C01430=1022.350,226.446,-123.530,169.335,49.096,159.350
C01431=1022.344,226.198,-123.503,169.332,49.101,159.351
C01432=1022.337,225.949,-123.477,169.328,49.105,159.351
C01433=1022.332,225.701,-123.450,169.325,49.109,159.352
C01434=1022.325,225.452,-123.423,169.321,49.114,159.352
C01435=1022.319,225.204,-123.397,169.318,49.118,159.352
C01436=1022.312,224.955,-123.370,169.314,49.122,159.353
C01437=1022.306,224.706,-123.343,169.310,49.128,159.353
C01438=1022.299,224.458,-123.316,169.306,49.132,159.354
C01439=1022.293,224.210,-123.290,169.303,49.137,159.354
C01440=1022.288,223.962,-123.263,169.299,49.141,159.354
C01441=1022.280,223.713,-123.236,169.296,49.145,159.355
C01442=1022.275,223.465,-123.210,169.292,49.150,159.355
C01443=1022.268,223.216,-123.183,169.289,49.154,159.356
C01444=1022.262,222.967,-123.157,169.285,49.159,159.356
C01445=1022.255,222.718,-123.130,169.282,49.163,159.357
C01446=1022.249,222.470,-123.104,169.277,49.168,159.357
C01447=1022.243,222.222,-123.077,169.274,49.173,159.357
C01448=1022.237,221.973,-123.050,169.270,49.177,159.358
C01449=1022.230,221.725,-123.024,169.267,49.182,159.358
C01450=1022.224,221.476,-122.997,169.263,49.186,159.359
C01451=1022.218,221.227,-122.970,169.260,49.191,159.359
C01452=1022.212,220.979,-122.944,169.256,49.195,159.359
C01453=1022.205,220.730,-122.917,169.253,49.200,159.360
C01454=1022.199,220.482,-122.891,169.249,49.204,159.360
C01455=1022.194,220.266,-122.869,169.246,49.208,159.361
C01456=1022.188,220.050,-122.845,169.243,49.212,159.361
C01457=1022.183,219.834,-122.822,169.239,49.216,159.362
C01458=1022.178,219.618,-122.799,169.237,49.220,159.362
C01459=1022.172,219.402,-122.776,169.234,49.224,159.362
C01460=1022.167,219.187,-122.753,169.230,49.228,159.363
C01461=1022.162,218.971,-122.730,169.228,49.232,159.363
C01462=1022.155,218.755,-122.707,169.224,49.236,159.363
C01463=1022.150,218.506,-122.680,169.221,49.241,159.364
C01464=1022.143,218.258,-122.654,169.217,49.246,159.364
C01465=1022.137,218.009,-122.628,169.214,49.250,159.365
C01466=1022.131,217.761,-122.602,169.211,49.255,159.365
C01467=1022.124,217.513,-122.576,169.206,49.260,159.366
C01468=1022.118,217.264,-122.549,169.203,49.265,159.366
C01469=1022.111,217.015,-122.524,169.199,49.270,159.367
C01470=1022.105,216.767,-122.498,169.196,49.274,159.367
C01471=1022.099,216.518,-122.471,169.193,49.279,159.368
C01472=1022.092,216.269,-122.445,169.189,49.284,159.368
C01473=1022.086,216.021,-122.419,169.185,49.289,159.369
C01474=1022.080,215.773,-122.392,169.182,49.294,159.369
C01475=1022.074,215.524,-122.367,169.178,49.299,159.370
C01476=1022.067,215.275,-122.341,169.175,49.303,159.370
C01477=1022.061,215.027,-122.314,169.171,49.308,159.371
C01478=1022.055,214.778,-122.289,169.168,49.313,159.371
C01479=1022.048,214.529,-122.262,169.164,49.318,159.372
C01480=1022.042,214.280,-122.236,169.161,49.323,159.372
C01481=1022.036,214.032,-122.210,169.157,49.327,159.373
C01482=1022.029,213.784,-122.184,169.154,49.332,159.373
C01483=1022.024,213.535,-122.158,169.150,49.337,159.374
C01484=1022.017,213.287,-122.132,169.147,49.342,159.374
C01485=1022.010,213.038,-122.107,169.143,49.347,159.375
C01486=1022.005,212.790,-122.080,169.139,49.352,159.375
C01487=1021.998,212.541,-122.055,169.136,49.357,159.376
C01488=1021.991,212.292,-122.028,169.133,49.361,159.376
C01489=1021.986,212.043,-122.002,169.129,49.366,159.377
C01490=1021.979,211.795,-121.976,169.126,49.371,159.377
C01491=1021.973,211.546,-121.951,169.123,49.375,159.378
C01492=1021.967,211.298,-121.924,169.118,49.381,159.378
C01493=1021.961,211.049,-121.899,169.115,49.386,159.379
C01494=1021.954,210.801,-121.872,169.112,49.390,159.379
C01495=1021.949,210.552,-121.847,169.109,49.395,159.380
C01496=1021.942,210.304,-121.820,169.105,49.400,159.380
C01497=1021.936,210.055,-121.795,169.102,49.405,159.381
C01498=1021.929,209.807,-121.769,169.098,49.410,159.381
C01499=1021.924,209.558,-121.743,169.094,49.415,159.382
C01500=1021.918,209.309,-121.718,169.091,49.420,159.382
C01501=1021.910,209.060,-121.691,169.088,49.425,159.383
C01502=1021.904,208.812,-121.666,169.085,49.430,159.383
C01503=1021.898,208.563,-121.641,169.080,49.435,159.384
C01504=1021.892,208.315,-121.615,169.077,49.440,159.384
C01505=1021.885,208.066,-121.589,169.074,49.445,159.385
C01506=1021.880,207.817,-121.563,169.071,49.451,159.386
C01507=1021.873,207.569,-121.537,169.067,49.456,159.386
C01508=1021.867,207.321,-121.512,169.063,49.461,159.387
C01509=1021.860,207.071,-121.486,169.060,49.466,159.387
C01510=1021.854,206.823,-121.461,169.057,49.471,159.388
C01511=1021.848,206.575,-121.435,169.054,49.475,159.388
C01512=1021.841,206.326,-121.410,169.050,49.481,159.389
C01513=1021.835,206.077,-121.384,169.046,49.486,159.389
C01514=1021.829,205.829,-121.359,169.043,49.491,159.390
C01515=1021.824,205.614,-121.337,169.040,49.495,159.390
C01516=1021.818,205.401,-121.315,169.037,49.500,159.391
C01517=1021.813,205.187,-121.292,169.034,49.504,159.391
C01518=1021.807,204.974,-121.271,169.031,49.509,159.392
C01519=1021.802,204.759,-121.249,169.028,49.514,159.392
C01520=1021.796,204.545,-121.227,169.026,49.518,159.393
C01521=1021.791,204.331,-121.205,169.022,49.523,159.393
C01522=1021.763,203.081,-121.084,168.586,49.431,159.305
C01523=1021.757,202.833,-121.060,168.581,49.437,159.306
C01524=1021.751,202.584,-121.036,168.577,49.443,159.306
C01525=1021.746,202.335,-121.013,168.573,49.449,159.307
C01526=1021.741,202.087,-120.988,168.569,49.456,159.308
C01527=1021.735,201.838,-120.965,168.565,49.462,159.308
C01528=1021.730,201.589,-120.941,168.560,49.468,159.309
C01529=1021.725,201.340,-120.917,168.556,49.474,159.310
C01530=1021.719,201.092,-120.894,168.552,49.480,159.310
C01531=1021.714,200.843,-120.870,168.547,49.486,159.311
C01532=1021.709,200.594,-120.846,168.543,49.492,159.311
C01533=1021.704,200.345,-120.822,168.539,49.498,159.312
C01534=1021.698,200.096,-120.799,168.534,49.504,159.312
C01535=1021.692,199.847,-120.774,168.530,49.511,159.313
C01536=1021.687,199.598,-120.751,168.526,49.517,159.314
C01537=1021.681,199.349,-120.727,168.521,49.523,159.314
C01538=1021.676,199.100,-120.704,168.517,49.529,159.315
C01539=1021.670,198.851,-120.681,168.513,49.536,159.316
C01540=1021.664,198.603,-120.657,168.509,49.542,159.316
C01541=1021.659,198.354,-120.633,168.505,49.548,159.317
C01542=1021.653,198.105,-120.610,168.500,49.555,159.317
C01543=1021.647,197.857,-120.587,168.496,49.560,159.318
C01544=1021.642,197.608,-120.563,168.491,49.567,159.319
C01545=1021.637,197.359,-120.540,168.488,49.573,159.319
C01546=1021.632,197.109,-120.517,168.484,49.579,159.320
C01547=1021.626,196.861,-120.493,168.479,49.586,159.320
C01548=1021.620,196.612,-120.470,168.475,49.591,159.321
C01549=1021.615,196.363,-120.447,168.471,49.598,159.322
C01550=1021.609,196.114,-120.424,168.466,49.604,159.322
C01551=1021.603,195.865,-120.401,168.462,49.610,159.323
C01552=1021.598,195.617,-120.376,168.459,49.617,159.324
C01553=1021.592,195.368,-120.354,168.454,49.623,159.324
C01554=1021.587,195.119,-120.331,168.450,49.629,159.325
C01555=1021.582,194.870,-120.307,168.446,49.636,159.326
C01556=1021.576,194.621,-120.284,168.441,49.642,159.326
C01557=1021.571,194.373,-120.262,168.438,49.648,159.327
C01558=1021.565,194.124,-120.237,168.434,49.655,159.328
C01559=1021.560,193.875,-120.214,168.429,49.661,159.328
C01560=1021.555,193.626,-120.191,168.425,49.667,159.329
C01561=1021.549,193.377,-120.168,168.421,49.673,159.329
C01562=1021.543,193.128,-120.145,168.417,49.680,159.330
C01563=1021.538,192.879,-120.121,168.413,49.686,159.331
C01564=1021.533,192.631,-120.099,168.409,49.692,159.331
C01565=1021.527,192.382,-120.076,168.405,49.698,159.332
C01566=1021.522,192.133,-120.052,168.401,49.705,159.333
C01567=1021.517,191.884,-120.029,168.397,49.711,159.333
C01568=1021.511,191.635,-120.006,168.393,49.717,159.334
C01569=1021.506,191.386,-119.983,168.388,49.724,159.334
C01570=1021.500,191.137,-119.960,168.384,49.730,159.335
C01571=1021.495,190.888,-119.937,168.380,49.736,159.336
C01572=1021.490,190.639,-119.914,168.377,49.743,159.336
C01573=1021.484,190.390,-119.891,168.372,49.749,159.337
C01574=1021.479,190.141,-119.868,168.368,49.755,159.338
C01575=1021.474,189.892,-119.844,168.364,49.762,159.338
C01576=1021.469,189.644,-119.822,168.360,49.768,159.339
C01577=1021.463,189.395,-119.799,168.357,49.774,159.340
C01578=1021.458,189.146,-119.775,168.352,49.780,159.340
C01579=1021.452,188.897,-119.752,168.348,49.786,159.341
C01580=1021.447,188.649,-119.730,168.344,49.793,159.342
C01581=1021.442,188.400,-119.706,168.340,49.799,159.342
C01582=1021.436,188.151,-119.683,168.336,49.805,159.343
C01583=1021.431,187.869,-119.658,168.332,49.813,159.344
C01584=1021.425,187.587,-119.632,168.328,49.820,159.344
C01585=1021.418,187.306,-119.605,168.323,49.827,159.345
C01586=1021.413,187.024,-119.580,168.319,49.834,159.346
C01587=1021.407,186.775,-119.557,168.314,49.841,159.346
C01588=1021.402,186.527,-119.534,168.310,49.847,159.347
C01589=1021.397,186.278,-119.511,168.306,49.853,159.348
C01590=1021.391,186.029,-119.488,168.303,49.859,159.348
C01591=1021.386,185.780,-119.465,168.299,49.865,159.349
C01592=1021.381,185.531,-119.443,168.295,49.872,159.350
C01593=1021.376,185.282,-119.420,168.290,49.878,159.350
C01594=1021.370,185.033,-119.397,168.286,49.884,159.351
C01595=1021.366,184.784,-119.373,168.283,49.891,159.352
C01596=1021.360,184.535,-119.351,168.279,49.897,159.352
C01597=1021.355,184.287,-119.329,168.275,49.903,159.353
C01598=1021.350,184.037,-119.305,168.271,49.909,159.354
C01599=1021.344,183.789,-119.282,168.267,49.915,159.354
C01600=1021.339,183.540,-119.260,168.264,49.922,159.355
C01601=1021.335,183.290,-119.237,168.260,49.928,159.356
C01602=1021.329,183.042,-119.214,168.255,49.934,159.356
C01603=1021.324,182.793,-119.192,168.252,49.941,159.357
C01604=1021.319,182.544,-119.168,168.248,49.947,159.357
C01605=1021.313,182.295,-119.145,168.244,49.954,159.358
C01606=1021.308,182.046,-119.124,168.240,49.960,159.359
C01607=1021.303,181.796,-119.101,168.237,49.966,159.360
C01608=1021.297,181.548,-119.079,168.233,49.973,159.360
C01609=1021.292,181.299,-119.057,168.228,49.979,159.361
C01610=1021.286,181.050,-119.034,168.225,49.986,159.362
C01611=1021.280,180.801,-119.013,168.221,49.993,159.362
C01612=1021.275,180.552,-118.991,168.217,49.999,159.363
C01613=1021.269,180.303,-118.968,168.213,50.006,159.364
C01614=1021.263,180.054,-118.946,168.209,50.013,159.365
C01615=1021.258,179.805,-118.924,168.206,50.019,159.365
C01616=1021.253,179.556,-118.902,168.202,50.025,159.366
C01617=1021.247,179.308,-118.880,168.198,50.032,159.367
C01618=1021.242,179.058,-118.858,168.194,50.039,159.367
C01619=1021.236,178.809,-118.836,168.190,50.045,159.368
C01620=1021.231,178.560,-118.813,168.186,50.052,159.369
C01621=1021.225,178.311,-118.791,168.183,50.058,159.370
C01622=1021.220,178.062,-118.770,168.179,50.065,159.370
C01623=1021.215,177.813,-118.747,168.174,50.071,159.371
C01624=1021.209,177.565,-118.725,168.171,50.078,159.372
C01625=1021.203,177.316,-118.703,168.167,50.085,159.372
C01626=1021.198,177.066,-118.681,168.163,50.091,159.373
C01627=1021.192,176.818,-118.660,168.160,50.098,159.374
C01628=1021.187,176.568,-118.637,168.156,50.104,159.374
C01629=1021.182,176.320,-118.615,168.152,50.111,159.375
C01630=1021.176,176.071,-118.593,168.148,50.117,159.376
C01631=1021.171,175.822,-118.571,168.144,50.124,159.377
C01632=1021.165,175.572,-118.549,168.141,50.131,159.377
C01633=1021.160,175.324,-118.528,168.137,50.137,159.378
C01634=1021.154,175.074,-118.506,168.134,50.144,159.379
C01635=1021.150,174.825,-118.484,168.130,50.150,159.379
C01636=1021.143,174.577,-118.461,168.127,50.157,159.380
C01637=1021.138,174.328,-118.439,168.122,50.163,159.381
C01638=1021.133,174.079,-118.417,168.118,50.170,159.382
C01639=1021.127,173.830,-118.396,168.115,50.177,159.382
C01640=1021.122,173.580,-118.374,168.111,50.183,159.383
C01641=1021.117,173.332,-118.352,168.107,50.189,159.384
C01642=1021.111,173.083,-118.331,168.104,50.196,159.384
C01643=1021.106,172.834,-118.308,168.100,50.203,159.385
C01644=1021.101,172.585,-118.286,168.096,50.209,159.386
C01645=1021.095,172.336,-118.265,168.093,50.216,159.387
C01646=1021.090,172.087,-118.243,168.089,50.222,159.387
C01647=1021.083,171.805,-118.218,168.085,50.229,159.388
C01648=1021.078,171.523,-118.194,168.081,50.237,159.389
C01649=1021.072,171.240,-118.168,168.077,50.245,159.390
C01650=1021.066,170.958,-118.144,168.072,50.252,159.391
C01651=1021.061,170.710,-118.122,168.069,50.259,159.391
C01652=1021.055,170.460,-118.101,168.065,50.265,159.392
C01653=1021.050,170.212,-118.079,168.061,50.272,159.393
C01654=1021.045,169.962,-118.057,168.058,50.278,159.393
C01655=1021.039,169.713,-118.035,168.054,50.285,159.394
C01656=1021.034,169.465,-118.014,168.051,50.292,159.395
C01657=1021.029,169.215,-117.991,168.047,50.298,159.396
C01658=1021.023,168.967,-117.970,168.043,50.305,159.396
C01659=1021.018,168.718,-117.948,168.040,50.311,159.397
C01660=1021.013,168.468,-117.926,168.036,50.317,159.398
C01661=1021.007,168.220,-117.905,168.033,50.324,159.399
C01662=1021.003,167.971,-117.883,168.029,50.331,159.399
C01663=1020.997,167.721,-117.861,168.025,50.337,159.400
C01664=1020.992,167.473,-117.839,168.022,50.344,159.401
C01665=1020.987,167.224,-117.818,168.018,50.350,159.401
C01666=1020.981,166.974,-117.797,168.015,50.357,159.402
C01667=1020.976,166.726,-117.775,168.011,50.363,159.403
C01668=1020.971,166.477,-117.753,168.007,50.370,159.404
C01669=1020.966,166.228,-117.732,168.004,50.377,159.404
C01670=1020.960,165.979,-117.709,168.000,50.383,159.405
C01671=1020.956,165.729,-117.688,167.997,50.390,159.406
C01672=1020.950,165.481,-117.667,167.993,50.396,159.406
C01673=1020.945,165.231,-117.645,167.990,50.403,159.407
C01674=1020.940,164.982,-117.623,167.986,50.409,159.408
C01675=1020.934,164.734,-117.602,167.982,50.416,159.409
C01676=1020.930,164.484,-117.580,167.980,50.422,159.410
C01677=1020.924,164.235,-117.559,167.976,50.428,159.410
C01678=1020.919,163.986,-117.537,167.973,50.435,159.411
C01679=1020.914,163.738,-117.515,167.969,50.442,159.412
C01680=1020.909,163.489,-117.494,167.965,50.448,159.412
C01681=1020.904,163.240,-117.473,167.962,50.455,159.413
C01682=1020.899,162.990,-117.450,167.958,50.462,159.414
C01683=1020.893,162.742,-117.429,167.955,50.468,159.414
C01684=1020.888,162.492,-117.408,167.951,50.474,159.415
C01685=1020.883,162.244,-117.387,167.948,50.481,159.416
C01686=1020.878,161.995,-117.365,167.944,50.487,159.416
C01687=1020.873,161.745,-117.343,167.941,50.494,159.417
C01688=1020.867,161.496,-117.322,167.938,50.500,159.418
C01689=1020.863,161.247,-117.300,167.934,50.507,159.419
C01690=1020.858,160.998,-117.279,167.931,50.513,159.419
C01691=1020.853,160.750,-117.258,167.927,50.520,159.420
C01692=1020.848,160.501,-117.236,167.924,50.527,159.421
C01693=1020.842,160.251,-117.215,167.920,50.533,159.422
C01694=1020.837,160.002,-117.193,167.917,50.539,159.423
C01695=1020.832,159.753,-117.171,167.914,50.546,159.423
C01696=1020.827,159.504,-117.151,167.910,50.552,159.424
C01697=1020.822,159.255,-117.129,167.907,50.559,159.425
C01698=1020.818,159.006,-117.108,167.903,50.566,159.425
C01699=1020.812,158.757,-117.086,167.899,50.572,159.426
C01700=1020.806,158.508,-117.066,167.896,50.579,159.427
C01701=1020.801,158.259,-117.044,167.892,50.586,159.428
C01702=1020.795,158.010,-117.024,167.889,50.592,159.428
C01703=1020.791,157.760,-117.003,167.886,50.599,159.429
C01704=1020.785,157.512,-116.981,167.883,50.606,159.430
C01705=1020.780,157.263,-116.961,167.880,50.612,159.431
C01706=1020.774,157.013,-116.940,167.876,50.619,159.432
C01707=1020.769,156.765,-116.919,167.873,50.626,159.432
C01708=1020.763,156.515,-116.898,167.869,50.632,159.433
C01709=1020.759,156.266,-116.877,167.866,50.639,159.434
C01710=1020.753,156.017,-116.856,167.862,50.646,159.434
C01711=1020.748,155.735,-116.832,167.858,50.653,159.435
C01712=1020.741,155.452,-116.809,167.855,50.661,159.436
C01713=1020.735,155.170,-116.785,167.851,50.669,159.437
C01714=1020.729,154.888,-116.761,167.847,50.676,159.438
C01715=1020.724,154.639,-116.741,167.843,50.683,159.439
C01716=1020.718,154.390,-116.719,167.840,50.690,159.439
C01717=1020.713,154.141,-116.699,167.836,50.696,159.440
C01718=1020.709,153.892,-116.678,167.834,50.703,159.441
C01719=1020.703,153.642,-116.657,167.830,50.710,159.442
C01720=1020.697,153.393,-116.636,167.827,50.716,159.443
C01721=1020.692,153.144,-116.615,167.824,50.723,159.443
C01722=1020.687,152.895,-116.594,167.820,50.730,159.444
C01723=1020.681,152.646,-116.574,167.817,50.737,159.445
C01724=1020.676,152.397,-116.553,167.813,50.743,159.446
C01725=1020.671,152.148,-116.533,167.809,50.750,159.446
C01726=1020.666,151.899,-116.512,167.806,50.757,159.447
C01727=1020.660,151.650,-116.491,167.804,50.763,159.448
C01728=1020.655,151.401,-116.470,167.800,50.770,159.449
C01729=1020.650,151.152,-116.450,167.797,50.777,159.449
C01730=1020.644,150.903,-116.429,167.793,50.784,159.450
C01731=1020.639,150.654,-116.409,167.790,50.790,159.451
C01732=1020.634,150.404,-116.388,167.787,50.797,159.452
C01733=1020.629,150.155,-116.368,167.783,50.804,159.453
C01734=1020.623,149.906,-116.347,167.780,50.811,159.453
C01735=1020.618,149.657,-116.327,167.777,50.817,159.454
C01736=1020.613,149.408,-116.306,167.774,50.824,159.455
C01737=1020.608,149.159,-116.285,167.771,50.831,159.456
C01738=1020.602,148.910,-116.265,167.767,50.838,159.457
C01739=1020.597,148.661,-116.244,167.764,50.845,159.457
C01740=1020.592,148.411,-116.224,167.760,50.851,159.458
C01741=1020.587,148.162,-116.203,167.757,50.858,159.459
C01742=1020.581,147.913,-116.183,167.754,50.864,159.460
C01743=1020.576,147.664,-116.162,167.751,50.871,159.460
C01744=1020.571,147.415,-116.142,167.747,50.878,159.461
C01745=1020.566,147.166,-116.121,167.744,50.885,159.462
C01746=1020.560,146.917,-116.100,167.741,50.891,159.463
C01747=1020.555,146.668,-116.080,167.737,50.898,159.463
C01748=1020.550,146.418,-116.059,167.735,50.905,159.464
C01749=1020.544,146.170,-116.039,167.731,50.912,159.465
C01750=1020.539,145.921,-116.019,167.728,50.918,159.466
C01751=1020.533,145.671,-115.998,167.725,50.925,159.467
C01752=1020.528,145.422,-115.978,167.721,50.932,159.467
C01753=1020.523,145.173,-115.958,167.718,50.939,159.468
C01754=1020.517,144.924,-115.938,167.714,50.946,159.469
C01755=1020.512,144.675,-115.917,167.712,50.952,159.470
C01756=1020.507,144.425,-115.897,167.709,50.959,159.471
C01757=1020.502,144.176,-115.877,167.705,50.966,159.471
C01758=1020.496,143.928,-115.857,167.702,50.973,159.472
C01759=1020.491,143.678,-115.837,167.698,50.980,159.473
C01760=1020.486,143.429,-115.816,167.695,50.987,159.474
C01761=1020.480,143.180,-115.797,167.692,50.993,159.475
C01762=1020.475,142.931,-115.776,167.689,51.000,159.475
C01763=1020.469,142.682,-115.756,167.686,51.007,159.476
C01764=1020.464,142.433,-115.735,167.683,51.014,159.477
C01765=1020.459,142.183,-115.716,167.679,51.021,159.478
C01766=1020.453,141.934,-115.696,167.676,51.027,159.479
C01767=1020.449,141.686,-115.675,167.673,51.034,159.479
C01768=1020.443,141.436,-115.656,167.670,51.041,159.480
C01769=1020.438,141.187,-115.636,167.667,51.048,159.481
C01770=1020.432,140.938,-115.615,167.663,51.055,159.482
C01771=1020.427,140.688,-115.595,167.660,51.061,159.482
C01772=1020.421,140.439,-115.575,167.658,51.068,159.483
C01773=1020.416,140.190,-115.555,167.654,51.075,159.484
C01774=1020.412,139.941,-115.535,167.651,51.082,159.485
C01775=1020.406,139.659,-115.513,167.647,51.090,159.486
C01776=1020.399,139.377,-115.490,167.644,51.097,159.487
C01777=1020.394,139.094,-115.467,167.640,51.105,159.488
